// TwinCAT 3 PLC project LS21002
// ProgramVersion: 3.1.4023.0
// libraries:
//   Recipe Management, * (System)
//   SysMem, * (System)
//   Tc2_EtherCAT, * (Beckhoff Automation GmbH)
//   Tc2_Math, * (Beckhoff Automation GmbH)
//   Tc2_MC2, * (Beckhoff Automation GmbH)
//   Tc2_MC2_Drive, * (Beckhoff Automation GmbH)
//   Tc2_ModbusSrv, * (Beckhoff Automation GmbH)
//   Tc2_SPA, * (Beckhoff Automation GmbH)
//   Tc2_Standard, * (Beckhoff Automation GmbH)
//   Tc2_SUPS, * (Beckhoff Automation GmbH)
//   Tc2_System, * (Beckhoff Automation GmbH)
//   Tc2_TcpIp, * (Beckhoff Automation GmbH)
//   Tc2_Utilities, * (Beckhoff Automation GmbH)
//   Tc3_Module, * (Beckhoff Automation GmbH)
//   BASE,1.0.0.0,MEGA
// project tree:
//   DUTs/Camera/ DUT_CameraSend.TcDUT, DUT_CameraReceive.TcDUT, ST_CameraPara.TcDUT
//   DUTs/ DUT_NCIO.TcDUT, DUT_NCIO_1.TcDUT
//   DUTs/EPS Robot/ CmdRobot1.TcDUT, DUT_SysFromRobot1.TcDUT, DUT_SysToRobot1.TcDUT, stPutPartPosChoose.TcDUT, stTakePartPosChoose.TcDUT
//   DUTs/IO/ EL1889.TcDUT, EL2889.TcDUT
//   DUTs/Others/ DUT_Calibration.TcDUT, DUT_Sta.TcDUT, DUT_StaHistory.TcDUT, stEasyPumpsParamter.TcDUT, stWorkStatus.TcDUT, tDateAndTime.TcDUT
//   DUTs/PartData/ DUT_BeltLineFixture.TcDUT, DUT_LidChecking.TcDUT, DUT_MainlineFixture.TcDUT, DUT_PartFlag.TcDUT, DUT_PartStatus.TcDUT, DUT_PartStatus_1.TcDUT, DUT_Robot2.TcDUT, DUT_Process.TcDUT
//   DUTs/PartSequence/ tsPartSequence.TcDUT, tsSequence.TcDUT
//   DUTs/PC/ DUT_FomularData.TcDUT, DUT_PCReceive.TcDUT, DUT_PCSend.TcDUT, DUT_UploadProcessData.TcDUT
//   DUTs/Recipe/ DUT.TcDUT, ST_Thermostat.TcDUT
//   GVLs/ Common.TcGVL, GVL_Config.TcGVL, GVL_Robot.TcGVL, GVL_PC.TcGVL, GVL_Standard.TcGVL, GVL_System.TcGVL, GVL_UPS.TcGVL, IO.TcGVL
//   / PlcTask.TcTTO
//   POUs/001_Station/001_Mapping/ InputLink.TcPOU, OutputLink.TcPOU
//   POUs/001_Station/ S01_Loading.TcPOU, S02_LidInjecting.TcPOU, S03_LidChecking.TcPOU, S04_AluCovering.TcPOU, S05_Adjusting.TcPOU, S06_Cutting.TcPOU, S07_BoxCarrying.TcPOU, S08_MainLine.TcPOU, S09_CardCarrying.TcPOU, S10_BeltCarrying.TcPOU, S11_Packing.TcPOU, S12_PreLine.TcPOU, S13_Labeling.TcPOU, S14_LabelChecking.TcPOU, S15_NG.TcPOU, S16_Unloading.TcPOU
//   POUs/002_Machine/ CallStandard.TcPOU, CommWithPC.TcPOU, ControlMachine.TcPOU, LightsTest.TcPOU
//   POUs/003_FB/0000_FB_Alive/ FB_Alive.TcPOU
//   POUs/003_FB/0014_HITBOT/ HITBOT_ERROR.TcDUT, stCmdType.TcDUT, stHIBOTLocalPara.TcDUT, FB_ERG_20C.TcPOU, stDeviceStatus.TcDUT, stOper_Para.TcDUT, stReadPara.TcDUT, stRealPara.TcDUT, stSetPara.TcDUT
//   POUs/003_FB/0015_Functions/001_Parallel/ FC_ParallelFinished.TcPOU, FC_ParallelRequest.TcPOU
//   POUs/003_FB/0015_Functions/ FC_BubbleSort_Max.TcPOU, FC_BubbleSort_Min.TcPOU
//   POUs/003_FB/03_TURINRobotFB/DUTs/ CmdRobot.TcDUT, DUT_SysFromRobot.TcDUT, DUT_SysToRobot.TcDUT, ST_Sys_Para.TcDUT, ST_TURINROBOT_Data.TcDUT, TURIN_ERROR.TcDUT, TURIN_STATE.TcDUT, T_MaxString.TcDUT
//   POUs/003_FB/03_TURINRobotFB/ FB_TURINContorl.TcPOU
//   POUs/003_FB/0001_200Smart/ FB_Modbus_200Smart.TcPOU
//   POUs/003_FB/0001_200Smart/S7-200SMART/ DUT_200SMART.TcDUT (not stored)
//   POUs/003_FB/0002_Camera/ FB_Camera.TcPOU
//   POUs/003_FB/0003_EtherCATState/ FB_EtherCatSlaveMonitor.TcPOU (not stored)
//   POUs/003_FB/0004_FlowLine/ DUT_Motor.TcDUT (not stored), FB_FlowLine.TcPOU
//   POUs/003_FB/0005_EncoderCounter/ FB_Encoder.TcPOU (not stored)
//   POUs/003_FB/0006_ATV/ FB_ATV12.TcPOU
//   POUs/003_FB/0007_Vacuum/ FB_SmcVacuum.TcPOU
//   POUs/003_FB/05_StationFB/ E_State.TcDUT, FB_Station.TcPOU
//   POUs/003_FB/0008_LocalClient/ FB_LocalClient.TcPOU
//   POUs/003_FB/0009_MKC204C/DUTs/ MT_MCK_CMD.TcDUT, MT_MCK_ERROR.TcDUT, ST_DeviceOpe.TcDUT, ST_MCK_ParIn.TcDUT (not stored), ST_MCK_ParOut.TcDUT, ST_SysPar.TcDUT
//   POUs/003_FB/0009_MKC204C/ FB_MKC204C.TcPOU
//   POUs/003_FB/0010_LoadCell/ DUT_DeviceOpe.TcDUT, ST_LoadCell_Error.TcDUT (not stored), FB_LoadCell.TcPOU, FB_Modbus_Tcp.TcPOU, stModbusPara.TcDUT (not stored), ST_LoadCell_ParOut.TcDUT (not stored)
//   POUs/003_FB/0011_Cimcor/ FB_Cimcor_IZN10E.TcPOU
//   POUs/003_FB/0012_EasyPump/DUT/ PumpError.TcDUT, stEasyPumpHeadType.TcDUT, stEasyPumpHmi.TcDUT, stEasyPumpSoftType.TcDUT, stEasyPumpType.TcDUT, stOperType.TcDUT, st_EasyPump.TcDUT, ST_StepStatus.TcDUT, ST_LocalPara.TcDUT, ST_ReadPara.TcDUT, ST_SetPara.TcDUT
//   POUs/003_FB/0012_EasyPump/ FB_KF300.TcPOU
//   POUs/003_FB/0013_RGI_14_new/不带旋转的电动夹爪/ FB_RGI_14_Modbus.TcPOU
//   POUs/003_FB/0013_RGI_14_new/带旋转的电动夹爪/ FB_RGI_14_Modbus_1.TcPOU (not stored)
//   POUs/003_FB/100_test/12_BlinkFB/ FB_Blinker.TcPOU (not stored), ST_SysPulse.TcDUT (not stored)
//   POUs/003_FB/100_test/ FB_GetTime.TcPOU
//   POUs/003_FB/10_CylinderFB/ FB_Cylinder.TcPOU, ST_DataCylinder.TcDUT
//   POUs/003_FB/0013_RGI_14_new/ RGI_14_CMD.TcDUT (not stored), RGI_14_ERROR.TcDUT, ST_RGI_14_IOData.TcDUT (not stored), ST_RGI_14_Sys_Para.TcDUT, ST_RGI_HMIStates.TcDUT, ST_RGI_Opera.TcDUT, ST_RGI_PosPara.TcDUT
//   POUs/003_FB/14_MachineFB/ FB_Machine.TcPOU, ST_DataMachine.TcDUT, ST_OpeButton.TcDUT
//   POUs/003_FB/17_HMIFB/ FB_Proface.TcPOU
//   POUs/003_FB/19-AxisFB/ DUT_ActPos.TcDUT, FB_Axis.TcPOU, FB_AxisHome.TcPOU, FB_Axis_old.TcPOU, ST_DataAxis.TcDUT
//   POUs/003_FB/41_GetSystemTime/ DUT_TIMESET.TcDUT, PRG_GetSystemTime.TcPOU
//   POUs/003_FB/43_implicit checks/ CheckBounds.TcPOU, CheckDivDInt.TcPOU, CheckDivLInt.TcPOU, CheckDivLReal.TcPOU, CheckDivReal.TcPOU, CheckLRangeSigned.TcPOU, CheckLRangeUnsigned.TcPOU, CheckPointer.TcPOU, CheckRangeSigned.TcPOU, CheckRangeUnsigned.TcPOU
//   POUs/003_FB/0016_Recipe/ FB_Recipes.TcPOU (not stored), ST_Recipe.TcDUT
//   POUs/003_FB/064_Temperature/ FB_TempControl_FUSHI.TcPOU, ST_FUSHI_PXF_ParRead.TcDUT (not stored), ST_FUSHI_PXF_ParSet.TcDUT (not stored), ST_FUSHI_PXF_Sys_Pointer.TcDUT (not stored)
//   POUs/003_FB/53_RudongPump/08_PeristalticPumpFB/DUTs/ RudongPump_CMD.TcDUT, RudongPump_ERROR.TcDUT, RudongPump_IOData.TcDUT, RudongPump_Ope.TcDUT, RudongPump_PumpHeadType.TcDUT, RudongPump_PumpType.TcDUT, RudongPump_RunData.TcDUT, RudongPump_SoftPipeType.TcDUT, RudongPump_Sys_Para.TcDUT, STATE_1.TcDUT, ST_ModbusAddress.TcDUT
//   POUs/003_FB/53_RudongPump/08_PeristalticPumpFB/ FB_RuDongPump_modbus_DF600Plus.TcPOU, FB_RuDongPump_modbus_LABV.TcPOU
//   POUs/003_FB/53_RudongPump/08_PeristalticPumpFB/校准程序/ AutoCal_CMD.TcDUT, AutoCal_ERROR.TcDUT, FB_AutoCal.TcPOU, STAutoCal_ParIn.TcDUT, STAutoCal_ParOut.TcDUT, ST_AutoCalOpe.TcDUT, ST_AutoCal_SysPar.TcDUT
//   POUs/003_FB/53_RudongPump/08_PeristalticPumpFB/梅特勒托利多秤/ FB_MT_MKC.TcPOU
//   POUs/003_FB/53_RudongPump/09_PeristalticPumpFB/ FB_RuDongPump_ModbusTCP.TcPOU, RudongPump_CMD_1.TcDUT, RudongPump_ERROR_1.TcDUT, RudongPump_IOData_1.TcDUT, RuDongPump_ModbusAddress.TcDUT, RudongPump_Ope_1.TcDUT, RudongPump_PumpHeadType_1.TcDUT, RudongPump_PumpType_1.TcDUT, RudongPump_RunData_1.TcDUT, RudongPump_SoftPipeType_1.TcDUT, RudongPump_Sys_Para_1.TcDUT
//   POUs/003_FB/53_RudongPump/41 Modbus指令/DataExchange/ ModbusTCP_ErrorQuery.TcPOU
//   POUs/003_FB/53_RudongPump/41 Modbus指令/ FB_ModbusTCP.TcPOU, ModbusParIn.TcDUT, ModbusParOut.TcDUT, Modbus_Cmd.TcDUT, Modbus_ErrorCode.TcDUT, Modbus_Operation.TcDUT, Modbus_SysPar.TcDUT
//   POUs/003_FB/Z_ERG_20 FB/DUTs/ ERG_20_CMD.TcDUT, ERG_20_ERROR.TcDUT, ST_ERG_20_IOData.TcDUT, ST_ERG_20_Sys_Para.TcDUT, ST_Huiling_Pers_Para.TcDUT, ST_Huiling_PosPara.TcDUT
//   POUs/003_FB/Z_ERG_20 FB/ FB_ERG_20_Modbus.TcPOU
//   POUs/40_TcpIp/40_TcpIp/ E_ClientSteps.TcDUT, E_DataExchaSteps.TcDUT (not stored), FB_ClientDataExcha.TcPOU, FB_TcpIpClient.TcPOU (not stored), stTcpIpBaseParaCfg.TcDUT (not stored), TcpIpClientConstants.TcGVL
//   POUs/ MAIN.TcPOU, RecipeManager.TcRMO (not stored)
// real-time tasks:
//   TASK PlcTask: cycle T#10ms, priority 20, ADS port 350
// motion (NC):
//   TASK NC-Task 1 SAF: cycle T#2ms, priority 4, ADS port 501
//   TASK NC-Task 1 SVB: cycle T#10ms, priority 8, ADS port 511
//   AXIS Axis 1 (id 1)
//     PositionAreaControl: Enable=false
//     TargetPosControl: Enable=false
//     OtherSettings: AllowMotionCmdToSlave=true
//     encoder EncType=19
//       EncPara: ScaleFactorNumerator=20, ScaleFactorDenominator=4194304, MaxCount=#xffffffff
//     drive DrvType=16
//       DrvPara: MaxCount=#xffffffff, DriveControlDWord=#x00020100
//         Analog: TorqueSetpointScale=10, ScaleFactorActTorque=0.1
//         TimeComp: TaskDelayCycles=1
//     controller CtrType=1
//       CtrPara: PriorControlFactor=1
//         PosDiffControl: Enable=false
//         Observer: BandWidth=20
//   AXIS Axis 2 (id 2)
//     PositionAreaControl: Enable=false
//     TargetPosControl: Enable=false
//     OtherSettings: AllowMotionCmdToSlave=true
//     encoder EncType=19
//       EncPara: ScaleFactorNumerator=20, ScaleFactorDenominator=4194304, MaxCount=#xffffffff
//     drive DrvType=16
//       DrvPara: MaxCount=#xffffffff, DriveControlDWord=#x00020100
//         Analog: TorqueSetpointScale=10, ScaleFactorActTorque=0.1
//         TimeComp: TaskDelayCycles=1
//     controller CtrType=1
//       CtrPara: PriorControlFactor=1
//         PosDiffControl: Enable=false
//         Observer: BandWidth=20
//   AXIS Axis 3 (id 3)
//     PositionAreaControl: Enable=false
//     TargetPosControl: Enable=false
//     OtherSettings: AllowMotionCmdToSlave=true
//     encoder EncType=19
//       EncPara: ScaleFactorNumerator=20, ScaleFactorDenominator=4194304, MaxCount=#xffffffff
//     drive DrvType=16
//       DrvPara: MaxCount=#xffffffff, DriveControlDWord=#x00020100
//         Analog: TorqueSetpointScale=10, ScaleFactorActTorque=0.1
//         TimeComp: TaskDelayCycles=1
//     controller CtrType=1
//       CtrPara: PriorControlFactor=1
//         PosDiffControl: Enable=false
//         Observer: BandWidth=20
//   AXIS Axis 4 (id 4)
//     PositionAreaControl: Enable=false
//     TargetPosControl: Enable=false
//     OtherSettings: AllowMotionCmdToSlave=true
//     encoder EncType=19
//       EncPara: ScaleFactorNumerator=20, ScaleFactorDenominator=4194304, MaxCount=#xffffffff
//     drive DrvType=16
//       DrvPara: MaxCount=#xffffffff, DriveControlDWord=#x00020100
//         Analog: TorqueSetpointScale=10, ScaleFactorActTorque=0.1
//         TimeComp: TaskDelayCycles=1
//     controller CtrType=1
//       CtrPara: PriorControlFactor=1
//         PosDiffControl: Enable=false
//         Observer: BandWidth=20
//   AXIS Axis 5 (id 5)
//     PositionAreaControl: Enable=false
//     TargetPosControl: Enable=false
//     OtherSettings: AllowMotionCmdToSlave=true
//     encoder EncType=19
//       EncPara: ScaleFactorNumerator=5, ScaleFactorDenominator=4194304, MaxCount=#xffffffff
//     drive DrvType=16
//       DrvPara: MaxCount=#xffffffff, DriveControlDWord=#x00020100
//         Analog: TorqueSetpointScale=10, ScaleFactorActTorque=0.1
//         TimeComp: TaskDelayCycles=1
//     controller CtrType=1
//       CtrPara: PriorControlFactor=1
//         PosDiffControl: Enable=false
//         Observer: BandWidth=20
//   AXIS Axis 6 (id 6)
//     PositionAreaControl: Enable=false
//     TargetPosControl: Enable=false
//     OtherSettings: AllowMotionCmdToSlave=true
//     encoder EncType=19
//       EncPara: ScaleFactorNumerator=20, ScaleFactorDenominator=4194304, MaxCount=#xffffffff
//     drive DrvType=16
//       DrvPara: MaxCount=#xffffffff, DriveControlDWord=#x00020100
//         Analog: TorqueSetpointScale=10, ScaleFactorActTorque=0.1
//         TimeComp: TaskDelayCycles=1
//     controller CtrType=1
//       CtrPara: PriorControlFactor=1
//         PosDiffControl: Enable=false
//         Observer: BandWidth=20
//   AXIS Axis 7 (id 7)
//     PositionAreaControl: Enable=false
//     TargetPosControl: Enable=false
//     OtherSettings: AllowMotionCmdToSlave=true
//     encoder EncType=19
//       EncPara: ScaleFactorNumerator=20, ScaleFactorDenominator=4194304, MaxCount=#xffffffff
//     drive DrvType=16
//       DrvPara: MaxCount=#xffffffff, DriveControlDWord=#x00020100
//         Analog: TorqueSetpointScale=10, ScaleFactorActTorque=0.1
//         TimeComp: TaskDelayCycles=1
//     controller CtrType=1
//       CtrPara: PriorControlFactor=1
//         PosDiffControl: Enable=false
//         Observer: BandWidth=20
//   AXIS Axis 8 (id 8)
//     PositionAreaControl: Enable=false
//     TargetPosControl: Enable=false
//     OtherSettings: AllowMotionCmdToSlave=true
//     encoder EncType=19
//       EncPara: ScaleFactorNumerator=5, ScaleFactorDenominator=4194304, MaxCount=#xffffffff
//     drive DrvType=16
//       DrvPara: MaxCount=#xffffffff, DriveControlDWord=#x00020100
//         Analog: TorqueSetpointScale=10, ScaleFactorActTorque=0.1
//         TimeComp: TaskDelayCycles=1
//     controller CtrType=1
//       CtrPara: PriorControlFactor=1
//         PosDiffControl: Enable=false
//         Observer: BandWidth=20
//   AXIS Axis 9 (id 9)
//     PositionAreaControl: Enable=false
//     TargetPosControl: Enable=false
//     OtherSettings: AllowMotionCmdToSlave=true
//     encoder EncType=19
//       EncPara: ScaleFactorNumerator=18, ScaleFactorDenominator=4194304, MaxCount=#xffffffff
//     drive DrvType=16
//       DrvPara: MaxCount=#xffffffff, DriveControlDWord=#x00020100
//         Analog: TorqueSetpointScale=10, ScaleFactorActTorque=0.1
//         TimeComp: TaskDelayCycles=1
//     controller CtrType=1
//       CtrPara: PriorControlFactor=1
//         PosDiffControl: Enable=false
//         Observer: BandWidth=20
//   AXIS Axis 10 (id 10)
//     PositionAreaControl: Enable=false
//     TargetPosControl: Enable=false
//     OtherSettings: AllowMotionCmdToSlave=true
//     encoder EncType=19
//       EncPara: ScaleFactorNumerator=2, ScaleFactorDenominator=4194304, MaxCount=#xffffffff
//     drive DrvType=16
//       DrvPara: MaxCount=#xffffffff, DriveControlDWord=#x00020100
//         Analog: TorqueSetpointScale=10, ScaleFactorActTorque=0.1
//         TimeComp: TaskDelayCycles=1
//     controller CtrType=1
//       CtrPara: PriorControlFactor=1
//         PosDiffControl: Enable=false
//         Observer: BandWidth=20
//   AXIS Axis 11 (id 11)
//     PositionAreaControl: Enable=false
//     TargetPosControl: Enable=false
//     OtherSettings: AllowMotionCmdToSlave=true
//     encoder EncType=19
//       EncPara: ScaleFactorNumerator=2, ScaleFactorDenominator=4194304, MaxCount=#xffffffff
//     drive DrvType=16
//       DrvPara: MaxCount=#xffffffff, DriveControlDWord=#x00020100
//         Analog: TorqueSetpointScale=10, ScaleFactorActTorque=0.1
//         TimeComp: TaskDelayCycles=1
//     controller CtrType=1
//       CtrPara: PriorControlFactor=1
//         PosDiffControl: Enable=false
//         Observer: BandWidth=20
//   AXIS Axis 12 (id 12)
//     PositionAreaControl: Enable=false
//     TargetPosControl: Enable=false
//     OtherSettings: AllowMotionCmdToSlave=true
//     encoder EncType=19
//       EncPara: ScaleFactorNumerator=2, ScaleFactorDenominator=4194304, MaxCount=#xffffffff
//     drive DrvType=16
//       DrvPara: MaxCount=#xffffffff, DriveControlDWord=#x00020100
//         Analog: TorqueSetpointScale=10, ScaleFactorActTorque=0.1
//         TimeComp: TaskDelayCycles=1
//     controller CtrType=1
//       CtrPara: PriorControlFactor=1
//         PosDiffControl: Enable=false
//         Observer: BandWidth=20
//   AXIS Axis 13 (id 13)
//     PositionAreaControl: Enable=false
//     TargetPosControl: Enable=false
//     OtherSettings: AllowMotionCmdToSlave=true
//     encoder EncType=19
//       EncPara: ScaleFactorNumerator=2, ScaleFactorDenominator=4194304, MaxCount=#xffffffff
//     drive DrvType=16
//       DrvPara: MaxCount=#xffffffff, DriveControlDWord=#x00020100
//         Analog: TorqueSetpointScale=10, ScaleFactorActTorque=0.1
//         TimeComp: TaskDelayCycles=1
//     controller CtrType=1
//       CtrPara: PriorControlFactor=1
//         PosDiffControl: Enable=false
//         Observer: BandWidth=20
//   AXIS Axis 14 (id 14)
//     PositionAreaControl: Enable=false
//     TargetPosControl: Enable=false
//     OtherSettings: AllowMotionCmdToSlave=true
//     encoder EncType=19
//       EncPara: ScaleFactorNumerator=36, ScaleFactorDenominator=4194304, MaxCount=#xffffffff
//     drive DrvType=16
//       DrvPara: MaxCount=#xffffffff, DriveControlDWord=#x00020100
//         Analog: TorqueSetpointScale=10, ScaleFactorActTorque=0.1
//         TimeComp: TaskDelayCycles=1
//     controller CtrType=1
//       CtrPara: PriorControlFactor=1
//         PosDiffControl: Enable=false
//         Observer: BandWidth=20
//   AXIS Axis 15 (id 15)
//     PositionAreaControl: Enable=false
//     TargetPosControl: Enable=false
//     OtherSettings: AllowMotionCmdToSlave=true
//     encoder EncType=19
//       EncPara: ScaleFactorNumerator=18.22123708, ScaleFactorDenominator=4194304, MaxCount=#xffffffff
//     drive DrvType=16
//       DrvPara: MaxCount=#xffffffff, DriveControlDWord=#x00020100
//         Analog: TorqueSetpointScale=10, ScaleFactorActTorque=0.1
//         TimeComp: TaskDelayCycles=1
//     controller CtrType=1
//       CtrPara: PriorControlFactor=1
//         PosDiffControl: Enable=false
//         Observer: BandWidth=20
//   AXIS Axis 16 (id 16)
//     PositionAreaControl: Enable=false
//     TargetPosControl: Enable=false
//     OtherSettings: AllowMotionCmdToSlave=true
//     encoder EncType=19
//       EncPara: ScaleFactorNumerator=20, ScaleFactorDenominator=4194304, MaxCount=#xffffffff
//     drive DrvType=16
//       DrvPara: MaxCount=#xffffffff, DriveControlDWord=#x00020100
//         Analog: TorqueSetpointScale=10, ScaleFactorActTorque=0.1
//         TimeComp: TaskDelayCycles=1
//     controller CtrType=1
//       CtrPara: PriorControlFactor=1
//         PosDiffControl: Enable=false
//         Observer: BandWidth=20
//   AXIS Axis 17 (id 17)
//     PositionAreaControl: Enable=false
//     TargetPosControl: Enable=false
//     OtherSettings: AllowMotionCmdToSlave=true
//     encoder EncType=19
//       EncPara: ScaleFactorNumerator=10, ScaleFactorDenominator=12800, MaxCount=#xffffffff
//     drive DrvType=16
//       DrvPara: MaxCount=#xffffffff, DriveControlDWord=#x00020000
//         Analog: TorqueSetpointScale=10, ScaleFactorActTorque=0.1
//         TimeComp: TaskDelayCycles=1
//     controller CtrType=1
//       CtrPara: PriorControlFactor=1
//         PosDiffControl: Enable=false
//         Observer: BandWidth=20
//   AXIS Axis 18 (id 18)
//     PositionAreaControl: Enable=false
//     TargetPosControl: Enable=false
//     OtherSettings: AllowMotionCmdToSlave=true
//     encoder EncType=19
//       EncPara: ScaleFactorNumerator=10, ScaleFactorDenominator=12800, MaxCount=#xffffffff
//     drive DrvType=16
//       DrvPara: MaxCount=#xffffffff, DriveControlDWord=#x00020000
//         Analog: TorqueSetpointScale=10, ScaleFactorActTorque=0.1
//         TimeComp: TaskDelayCycles=1
//     controller CtrType=1
//       CtrPara: PriorControlFactor=1
//         PosDiffControl: Enable=false
//         Observer: BandWidth=20
//   AXIS Axis 19 (id 19)
//     PositionAreaControl: Enable=false
//     TargetPosControl: Enable=false
//     OtherSettings: AllowMotionCmdToSlave=true
//     encoder EncType=19
//       EncPara: ScaleFactorNumerator=10, ScaleFactorDenominator=12800, MaxCount=#xffffffff
//     drive DrvType=16
//       DrvPara: MaxCount=#xffffffff, DriveControlDWord=#x00020000
//         Analog: TorqueSetpointScale=10, ScaleFactorActTorque=0.1
//         TimeComp: TaskDelayCycles=1
//     controller CtrType=1
//       CtrPara: PriorControlFactor=1
//         PosDiffControl: Enable=false
//         Observer: BandWidth=20
// I/O:
//   DEVICE Device 1 (EtherCAT), AmsNetId 192.168.1.1.2.1
//     Term 16 (EK1200) [EK1200-5000 EtherCAT Power supply (2A E-Bus)]
//       Term 2 (EL1889) [EL1889 16Ch. Dig. Input 24V, 3ms, negative]
//       Term 3 (EL1889) [EL1889 16Ch. Dig. Input 24V, 3ms, negative]
//       Term 4 (EL1889) [EL1889 16Ch. Dig. Input 24V, 3ms, negative]
//       Term 5 (EL1889) [EL1889 16Ch. Dig. Input 24V, 3ms, negative]
//       Term 6 (EL1889) [EL1889 16Ch. Dig. Input 24V, 3ms, negative]
//       Term 7 (EL1889) [EL1889 16Ch. Dig. Input 24V, 3ms, negative]
//       Term 8 (EL2889) [EL2889 16Ch. Dig. Output 24V, 0.5A, negative]
//       Term 9 (EL2889) [EL2889 16Ch. Dig. Output 24V, 0.5A, negative]
//       Term 25 (EL2889) [EL2889 16Ch. Dig. Output 24V, 0.5A, negative]
//       Term 26 (EL2889) [EL2889 16Ch. Dig. Output 24V, 0.5A, negative]
//       Term 27 (EL2889) [EL2889 16Ch. Dig. Output 24V, 0.5A, negative]
//       Term 28 (EL2889) [EL2889 16Ch. Dig. Output 24V, 0.5A, negative]
//       Term 29 (EK1122) [EK1122 2 port EtherCAT junction]
//         Drive 30 (MR-JET-G-N1) [MR-JET-G-N1 EtherCAT Drive (CoE) ver.B9]
//         Drive 31 (MR-JET-G-N1) [MR-JET-G-N1 EtherCAT Drive (CoE) ver.B9]
//         Drive 32 (MR-JET-G-N1) [MR-JET-G-N1 EtherCAT Drive (CoE) ver.B9]
//         Drive 33 (MR-JET-G-N1) [MR-JET-G-N1 EtherCAT Drive (CoE) ver.B9]
//         Drive 34 (MR-JET-G-N1) [MR-JET-G-N1 EtherCAT Drive (CoE) ver.C0]
//         Drive 35 (MR-JET-G-N1) [MR-JET-G-N1 EtherCAT Drive (CoE) ver.B9]
//         Drive 36 (MR-JET-G-N1) [MR-JET-G-N1 EtherCAT Drive (CoE) ver.B9]
//         Drive 37 (MR-JET-G-N1) [MR-JET-G-N1 EtherCAT Drive (CoE) ver.C0]
//         Term 38 (EK1100) [EK1100 EtherCAT Coupler (2A E-Bus)]
//           Term 39 (EL1889) [EL1889 16Ch. Dig. Input 24V, 3ms, negative]
//           Term 73 (EL2889) [EL2889 16Ch. Dig. Output 24V, 0.5A, negative]
//           Term 62 (EL9011) [EL9011 End Terminal]
//         Drive 40 (MR-JET-G-N1) [MR-JET-G-N1 EtherCAT Drive (CoE) ver.B9]
//         Term 41 (EK1100) [EK1100 EtherCAT Coupler (2A E-Bus)]
//           Term 42 (EL1889) [EL1889 16Ch. Dig. Input 24V, 3ms, negative]
//           Term 43 (EL1889) [EL1889 16Ch. Dig. Input 24V, 3ms, negative]
//           Term 44 (EL1889) [EL1889 16Ch. Dig. Input 24V, 3ms, negative]
//           Term 45 (EL1889) [EL1889 16Ch. Dig. Input 24V, 3ms, negative]
//           Term 46 (EL1889) [EL1889 16Ch. Dig. Input 24V, 3ms, negative]
//           Term 47 (EL1889) [EL1889 16Ch. Dig. Input 24V, 3ms, negative]
//           Term 48 (EL2889) [EL2889 16Ch. Dig. Output 24V, 0.5A, negative]
//           Term 49 (EL2889) [EL2889 16Ch. Dig. Output 24V, 0.5A, negative]
//           Term 50 (EL2889) [EL2889 16Ch. Dig. Output 24V, 0.5A, negative]
//           Term 51 (EL2889) [EL2889 16Ch. Dig. Output 24V, 0.5A, negative]
//           Term 63 (EL9011) [EL9011 End Terminal]
//         Drive 52 (MR-JET-G-N1) [MR-JET-G-N1 EtherCAT Drive (CoE) ver.C0]
//         Drive 53 (MR-JET-G-N1) [MR-JET-G-N1 EtherCAT Drive (CoE) ver.C0]
//         Drive 54 (MR-JET-G-N1) [MR-JET-G-N1 EtherCAT Drive (CoE) ver.C0]
//         Drive 55 (MR-JET-G-N1) [MR-JET-G-N1 EtherCAT Drive (CoE) ver.C0]
//         Drive 56 (MR-JET-G-N1) [MR-JET-G-N1 EtherCAT Drive (CoE) ver.C0]
//         Drive 57 (MR-JET-G-N1) [MR-JET-G-N1 EtherCAT Drive (CoE) ver.C0]
//         Drive 58 (MR-JET-G-N1) [MR-JET-G-N1 EtherCAT Drive (CoE) ver.B9]
//         Drive 59 (DM3C-EC556) [DM3C-EC556(COE)]
//         Drive 60 (DM3C-EC556) [DM3C-EC556(COE)]
//         Drive 61 (DM3C-EC870) [DM3C-EC870(COE)]
//         Term 95 (EK1100) [EK1100 EtherCAT Coupler (2A E-Bus)]
//           Term 96 (EL1889) [EL1889 16Ch. Dig. Input 24V, 3ms, negative]
//           Term 97 (EL1889) [EL1889 16Ch. Dig. Input 24V, 3ms, negative]
//           Term 98 (EL2889) [EL2889 16Ch. Dig. Output 24V, 0.5A, negative]
//           Term 99 (EL2889) [EL2889 16Ch. Dig. Output 24V, 0.5A, negative]
//           Term 103 (EL9011) [EL9011 End Terminal]
//         Box 100 (GR10-2HCE) [GR10-2HCE_1.4.5.0]
//   DEVICE Device 2 (EtherCAT Automation Protocol), AmsNetId 192.168.1.1.3.1
//   DEVICE Device 3 (EtherCAT Automation Protocol), AmsNetId 192.168.1.1.4.1
//   DEVICE Device 4 (COM Port)
// variable links:
//   NC-Task 1 SAF/Axes/Axis 1 <-> Device 1 (EtherCAT)/Term 16 (EK1200)/Term 29 (EK1122)/Drive 30 (MR-JET-G-N1)
//     Drive/Inputs/In/nDataIn1 <-> 1st Transmit PDO Mapping/Following error actual value
//     Drive/Inputs/In/nDataIn3[0] <-> 1st Transmit PDO Mapping/Torque actual value
//     Drive/Inputs/In/nDcOutputTime <-> InfoData/DcOutputShift
//     Drive/Inputs/In/nState1 <-> 1st Transmit PDO Mapping/Statusword
//     Drive/Inputs/In/nState2 <-> 1st Transmit PDO Mapping/Statusword @bit 8
//     Drive/Inputs/In/nState4 @bit 1 <-> WcState/InputToggle
//     Drive/Inputs/In/nState4 <-> WcState/WcState
//     Drive/Inputs/In/nState5 <-> 1st Transmit PDO Mapping/Modes of operation display
//     Drive/Outputs/Out/nDataOut1 <-> 1st Receive PDO Mapping/Target position
//     Drive/Outputs/Out/nDataOut2 <-> 1st Receive PDO Mapping/Target velocity
//     Drive/Outputs/Out/nDataOut4[0] <-> 1st Receive PDO Mapping/Target torque
//     Enc/Inputs/In/nDataIn1 <-> 1st Transmit PDO Mapping/Position actual value
//     Enc/Inputs/In/nDataIn7 <-> 1st Transmit PDO Mapping/Velocity actual value
//     Enc/Inputs/In/nDcInputTime <-> InfoData/DcInputShift
//     Enc/Inputs/In/nState4 @bit 1 <-> WcState/InputToggle
//     Enc/Inputs/In/nState4 <-> WcState/WcState
//   NC-Task 1 SAF/Axes/Axis 10 <-> Device 1 (EtherCAT)/Term 16 (EK1200)/Term 29 (EK1122)/Drive 52 (MR-JET-G-N1)
//     Drive/Inputs/In/nDataIn1 <-> 1st Transmit PDO Mapping/Following error actual value
//     Drive/Inputs/In/nDataIn3[0] <-> 1st Transmit PDO Mapping/Torque actual value
//     Drive/Inputs/In/nDcOutputTime <-> InfoData/DcOutputShift
//     Drive/Inputs/In/nState1 <-> 1st Transmit PDO Mapping/Statusword
//     Drive/Inputs/In/nState2 <-> 1st Transmit PDO Mapping/Statusword @bit 8
//     Drive/Inputs/In/nState4 @bit 1 <-> WcState/InputToggle
//     Drive/Inputs/In/nState4 <-> WcState/WcState
//     Drive/Inputs/In/nState5 <-> 1st Transmit PDO Mapping/Modes of operation display
//     Drive/Outputs/Out/nDataOut1 <-> 1st Receive PDO Mapping/Target position
//     Drive/Outputs/Out/nDataOut2 <-> 1st Receive PDO Mapping/Target velocity
//     Drive/Outputs/Out/nDataOut4[0] <-> 1st Receive PDO Mapping/Target torque
//     Enc/Inputs/In/nDataIn1 <-> 1st Transmit PDO Mapping/Position actual value
//     Enc/Inputs/In/nDataIn7 <-> 1st Transmit PDO Mapping/Velocity actual value
//     Enc/Inputs/In/nDcInputTime <-> InfoData/DcInputShift
//     Enc/Inputs/In/nState4 @bit 1 <-> WcState/InputToggle
//     Enc/Inputs/In/nState4 <-> WcState/WcState
//   NC-Task 1 SAF/Axes/Axis 11 <-> Device 1 (EtherCAT)/Term 16 (EK1200)/Term 29 (EK1122)/Drive 53 (MR-JET-G-N1)
//     Drive/Inputs/In/nDataIn1 <-> 1st Transmit PDO Mapping/Following error actual value
//     Drive/Inputs/In/nDataIn3[0] <-> 1st Transmit PDO Mapping/Torque actual value
//     Drive/Inputs/In/nDcOutputTime <-> InfoData/DcOutputShift
//     Drive/Inputs/In/nState1 <-> 1st Transmit PDO Mapping/Statusword
//     Drive/Inputs/In/nState2 <-> 1st Transmit PDO Mapping/Statusword @bit 8
//     Drive/Inputs/In/nState4 @bit 1 <-> WcState/InputToggle
//     Drive/Inputs/In/nState4 <-> WcState/WcState
//     Drive/Inputs/In/nState5 <-> 1st Transmit PDO Mapping/Modes of operation display
//     Drive/Outputs/Out/nDataOut1 <-> 1st Receive PDO Mapping/Target position
//     Drive/Outputs/Out/nDataOut2 <-> 1st Receive PDO Mapping/Target velocity
//     Drive/Outputs/Out/nDataOut4[0] <-> 1st Receive PDO Mapping/Target torque
//     Enc/Inputs/In/nDataIn1 <-> 1st Transmit PDO Mapping/Position actual value
//     Enc/Inputs/In/nDataIn7 <-> 1st Transmit PDO Mapping/Velocity actual value
//     Enc/Inputs/In/nDcInputTime <-> InfoData/DcInputShift
//     Enc/Inputs/In/nState4 @bit 1 <-> WcState/InputToggle
//     Enc/Inputs/In/nState4 <-> WcState/WcState
//   NC-Task 1 SAF/Axes/Axis 12 <-> Device 1 (EtherCAT)/Term 16 (EK1200)/Term 29 (EK1122)/Drive 54 (MR-JET-G-N1)
//     Drive/Inputs/In/nDataIn1 <-> 1st Transmit PDO Mapping/Following error actual value
//     Drive/Inputs/In/nDataIn3[0] <-> 1st Transmit PDO Mapping/Torque actual value
//     Drive/Inputs/In/nDcOutputTime <-> InfoData/DcOutputShift
//     Drive/Inputs/In/nState1 <-> 1st Transmit PDO Mapping/Statusword
//     Drive/Inputs/In/nState2 <-> 1st Transmit PDO Mapping/Statusword @bit 8
//     Drive/Inputs/In/nState4 @bit 1 <-> WcState/InputToggle
//     Drive/Inputs/In/nState4 <-> WcState/WcState
//     Drive/Inputs/In/nState5 <-> 1st Transmit PDO Mapping/Modes of operation display
//     Drive/Outputs/Out/nDataOut1 <-> 1st Receive PDO Mapping/Target position
//     Drive/Outputs/Out/nDataOut2 <-> 1st Receive PDO Mapping/Target velocity
//     Drive/Outputs/Out/nDataOut4[0] <-> 1st Receive PDO Mapping/Target torque
//     Enc/Inputs/In/nDataIn1 <-> 1st Transmit PDO Mapping/Position actual value
//     Enc/Inputs/In/nDataIn7 <-> 1st Transmit PDO Mapping/Velocity actual value
//     Enc/Inputs/In/nDcInputTime <-> InfoData/DcInputShift
//     Enc/Inputs/In/nState4 @bit 1 <-> WcState/InputToggle
//     Enc/Inputs/In/nState4 <-> WcState/WcState
//   NC-Task 1 SAF/Axes/Axis 13 <-> Device 1 (EtherCAT)/Term 16 (EK1200)/Term 29 (EK1122)/Drive 55 (MR-JET-G-N1)
//     Drive/Inputs/In/nDataIn1 <-> 1st Transmit PDO Mapping/Following error actual value
//     Drive/Inputs/In/nDataIn3[0] <-> 1st Transmit PDO Mapping/Torque actual value
//     Drive/Inputs/In/nDcOutputTime <-> InfoData/DcOutputShift
//     Drive/Inputs/In/nState1 <-> 1st Transmit PDO Mapping/Statusword
//     Drive/Inputs/In/nState2 <-> 1st Transmit PDO Mapping/Statusword @bit 8
//     Drive/Inputs/In/nState4 @bit 1 <-> WcState/InputToggle
//     Drive/Inputs/In/nState4 <-> WcState/WcState
//     Drive/Inputs/In/nState5 <-> 1st Transmit PDO Mapping/Modes of operation display
//     Drive/Outputs/Out/nDataOut1 <-> 1st Receive PDO Mapping/Target position
//     Drive/Outputs/Out/nDataOut2 <-> 1st Receive PDO Mapping/Target velocity
//     Drive/Outputs/Out/nDataOut4[0] <-> 1st Receive PDO Mapping/Target torque
//     Enc/Inputs/In/nDataIn1 <-> 1st Transmit PDO Mapping/Position actual value
//     Enc/Inputs/In/nDataIn7 <-> 1st Transmit PDO Mapping/Velocity actual value
//     Enc/Inputs/In/nDcInputTime <-> InfoData/DcInputShift
//     Enc/Inputs/In/nState4 @bit 1 <-> WcState/InputToggle
//     Enc/Inputs/In/nState4 <-> WcState/WcState
//   NC-Task 1 SAF/Axes/Axis 14 <-> Device 1 (EtherCAT)/Term 16 (EK1200)/Term 29 (EK1122)/Drive 56 (MR-JET-G-N1)
//     Drive/Inputs/In/nDataIn1 <-> 1st Transmit PDO Mapping/Following error actual value
//     Drive/Inputs/In/nDataIn3[0] <-> 1st Transmit PDO Mapping/Torque actual value
//     Drive/Inputs/In/nDcOutputTime <-> InfoData/DcOutputShift
//     Drive/Inputs/In/nState1 <-> 1st Transmit PDO Mapping/Statusword
//     Drive/Inputs/In/nState2 <-> 1st Transmit PDO Mapping/Statusword @bit 8
//     Drive/Inputs/In/nState4 @bit 1 <-> WcState/InputToggle
//     Drive/Inputs/In/nState4 <-> WcState/WcState
//     Drive/Inputs/In/nState5 <-> 1st Transmit PDO Mapping/Modes of operation display
//     Drive/Outputs/Out/nDataOut1 <-> 1st Receive PDO Mapping/Target position
//     Drive/Outputs/Out/nDataOut2 <-> 1st Receive PDO Mapping/Target velocity
//     Drive/Outputs/Out/nDataOut4[0] <-> 1st Receive PDO Mapping/Target torque
//     Enc/Inputs/In/nDataIn1 <-> 1st Transmit PDO Mapping/Position actual value
//     Enc/Inputs/In/nDataIn7 <-> 1st Transmit PDO Mapping/Velocity actual value
//     Enc/Inputs/In/nDcInputTime <-> InfoData/DcInputShift
//     Enc/Inputs/In/nState4 @bit 1 <-> WcState/InputToggle
//     Enc/Inputs/In/nState4 <-> WcState/WcState
//   NC-Task 1 SAF/Axes/Axis 15 <-> Device 1 (EtherCAT)/Term 16 (EK1200)/Term 29 (EK1122)/Drive 57 (MR-JET-G-N1)
//     Drive/Inputs/In/nDataIn1 <-> 1st Transmit PDO Mapping/Following error actual value
//     Drive/Inputs/In/nDataIn3[0] <-> 1st Transmit PDO Mapping/Torque actual value
//     Drive/Inputs/In/nDcOutputTime <-> InfoData/DcOutputShift
//     Drive/Inputs/In/nState1 <-> 1st Transmit PDO Mapping/Statusword
//     Drive/Inputs/In/nState2 <-> 1st Transmit PDO Mapping/Statusword @bit 8
//     Drive/Inputs/In/nState4 @bit 1 <-> WcState/InputToggle
//     Drive/Inputs/In/nState4 <-> WcState/WcState
//     Drive/Inputs/In/nState5 <-> 1st Transmit PDO Mapping/Modes of operation display
//     Drive/Outputs/Out/nDataOut1 <-> 1st Receive PDO Mapping/Target position
//     Drive/Outputs/Out/nDataOut2 <-> 1st Receive PDO Mapping/Target velocity
//     Drive/Outputs/Out/nDataOut4[0] <-> 1st Receive PDO Mapping/Target torque
//     Enc/Inputs/In/nDataIn1 <-> 1st Transmit PDO Mapping/Position actual value
//     Enc/Inputs/In/nDataIn7 <-> 1st Transmit PDO Mapping/Velocity actual value
//     Enc/Inputs/In/nDcInputTime <-> InfoData/DcInputShift
//     Enc/Inputs/In/nState4 @bit 1 <-> WcState/InputToggle
//     Enc/Inputs/In/nState4 <-> WcState/WcState
//   NC-Task 1 SAF/Axes/Axis 16 <-> Device 1 (EtherCAT)/Term 16 (EK1200)/Term 29 (EK1122)/Drive 58 (MR-JET-G-N1)
//     Drive/Inputs/In/nDataIn1 <-> 1st Transmit PDO Mapping/Following error actual value
//     Drive/Inputs/In/nDataIn3[0] <-> 1st Transmit PDO Mapping/Torque actual value
//     Drive/Inputs/In/nDcOutputTime <-> InfoData/DcOutputShift
//     Drive/Inputs/In/nState1 <-> 1st Transmit PDO Mapping/Statusword
//     Drive/Inputs/In/nState2 <-> 1st Transmit PDO Mapping/Statusword @bit 8
//     Drive/Inputs/In/nState4 @bit 1 <-> WcState/InputToggle
//     Drive/Inputs/In/nState4 <-> WcState/WcState
//     Drive/Inputs/In/nState5 <-> 1st Transmit PDO Mapping/Modes of operation display
//     Drive/Outputs/Out/nDataOut1 <-> 1st Receive PDO Mapping/Target position
//     Drive/Outputs/Out/nDataOut2 <-> 1st Receive PDO Mapping/Target velocity
//     Drive/Outputs/Out/nDataOut4[0] <-> 1st Receive PDO Mapping/Target torque
//     Enc/Inputs/In/nDataIn1 <-> 1st Transmit PDO Mapping/Position actual value
//     Enc/Inputs/In/nDataIn7 <-> 1st Transmit PDO Mapping/Velocity actual value
//     Enc/Inputs/In/nDcInputTime <-> InfoData/DcInputShift
//     Enc/Inputs/In/nState4 @bit 1 <-> WcState/InputToggle
//     Enc/Inputs/In/nState4 <-> WcState/WcState
//   NC-Task 1 SAF/Axes/Axis 17 <-> Device 1 (EtherCAT)/Term 16 (EK1200)/Term 29 (EK1122)/Drive 59 (DM3C-EC556)
//     Drive/Inputs/In/nDcOutputTime <-> InfoData/DcOutputShift
//     Drive/Inputs/In/nState1 <-> Transmit PDO 1/Status Word
//     Drive/Inputs/In/nState2 <-> Transmit PDO 1/Status Word @bit 8
//     Drive/Inputs/In/nState4 @bit 1 <-> WcState/InputToggle
//     Drive/Inputs/In/nState4 <-> WcState/WcState
//     Drive/Inputs/In/nState5 <-> Transmit PDO 1/Modes of Operation display
//     Drive/Outputs/Out/nDataOut1 <-> Receive PDO 1/Profile Target Position
//     Enc/Inputs/In/nDataIn1 <-> Transmit PDO 1/Position Actual Value
//     Enc/Inputs/In/nDataIn3 <-> Transmit PDO 1/Touch Probe 1 Positive Value
//     Enc/Inputs/In/nDcInputTime <-> InfoData/DcInputShift
//     Enc/Inputs/In/nState4 @bit 1 <-> WcState/InputToggle
//     Enc/Inputs/In/nState4 <-> WcState/WcState
//     Enc/Inputs/In/nState5 <-> Transmit PDO 1/Touch Probe Status
//     Enc/Inputs/In/nState6 <-> Transmit PDO 1/Touch Probe Status @bit 8
//     Enc/Outputs/Out/nCtrl5 <-> Receive PDO 1/Touch Probe Function
//     Enc/Outputs/Out/nCtrl6 <-> Receive PDO 1/Touch Probe Function @bit 8
//   NC-Task 1 SAF/Axes/Axis 18 <-> Device 1 (EtherCAT)/Term 16 (EK1200)/Term 29 (EK1122)/Drive 60 (DM3C-EC556)
//     Drive/Inputs/In/nDcOutputTime <-> InfoData/DcOutputShift
//     Drive/Inputs/In/nState1 <-> Transmit PDO 1/Status Word
//     Drive/Inputs/In/nState2 <-> Transmit PDO 1/Status Word @bit 8
//     Drive/Inputs/In/nState4 @bit 1 <-> WcState/InputToggle
//     Drive/Inputs/In/nState4 <-> WcState/WcState
//     Drive/Inputs/In/nState5 <-> Transmit PDO 1/Modes of Operation display
//     Drive/Outputs/Out/nDataOut1 <-> Receive PDO 1/Profile Target Position
//     Enc/Inputs/In/nDataIn1 <-> Transmit PDO 1/Position Actual Value
//     Enc/Inputs/In/nDataIn3 <-> Transmit PDO 1/Touch Probe 1 Positive Value
//     Enc/Inputs/In/nDcInputTime <-> InfoData/DcInputShift
//     Enc/Inputs/In/nState4 @bit 1 <-> WcState/InputToggle
//     Enc/Inputs/In/nState4 <-> WcState/WcState
//     Enc/Inputs/In/nState5 <-> Transmit PDO 1/Touch Probe Status
//     Enc/Inputs/In/nState6 <-> Transmit PDO 1/Touch Probe Status @bit 8
//     Enc/Outputs/Out/nCtrl5 <-> Receive PDO 1/Touch Probe Function
//     Enc/Outputs/Out/nCtrl6 <-> Receive PDO 1/Touch Probe Function @bit 8
//   NC-Task 1 SAF/Axes/Axis 19 <-> Device 1 (EtherCAT)/Term 16 (EK1200)/Term 29 (EK1122)/Drive 61 (DM3C-EC870)
//     Drive/Inputs/In/nDcOutputTime <-> InfoData/DcOutputShift
//     Drive/Inputs/In/nState1 <-> Transmit PDO 1/Status Word
//     Drive/Inputs/In/nState2 <-> Transmit PDO 1/Status Word @bit 8
//     Drive/Inputs/In/nState4 @bit 1 <-> WcState/InputToggle
//     Drive/Inputs/In/nState4 <-> WcState/WcState
//     Drive/Inputs/In/nState5 <-> Transmit PDO 1/Modes of Operation display
//     Drive/Outputs/Out/nDataOut1 <-> Receive PDO 1/Profile Target Position
//     Enc/Inputs/In/nDataIn1 <-> Transmit PDO 1/Position Actual Value
//     Enc/Inputs/In/nDataIn3 <-> Transmit PDO 1/Touch Probe 1 Positive Value
//     Enc/Inputs/In/nDcInputTime <-> InfoData/DcInputShift
//     Enc/Inputs/In/nState4 @bit 1 <-> WcState/InputToggle
//     Enc/Inputs/In/nState4 <-> WcState/WcState
//     Enc/Inputs/In/nState5 <-> Transmit PDO 1/Touch Probe Status
//     Enc/Inputs/In/nState6 <-> Transmit PDO 1/Touch Probe Status @bit 8
//     Enc/Outputs/Out/nCtrl5 <-> Receive PDO 1/Touch Probe Function
//     Enc/Outputs/Out/nCtrl6 <-> Receive PDO 1/Touch Probe Function @bit 8
//   NC-Task 1 SAF/Axes/Axis 2 <-> Device 1 (EtherCAT)/Term 16 (EK1200)/Term 29 (EK1122)/Drive 31 (MR-JET-G-N1)
//     Drive/Inputs/In/nDataIn1 <-> 1st Transmit PDO Mapping/Following error actual value
//     Drive/Inputs/In/nDataIn3[0] <-> 1st Transmit PDO Mapping/Torque actual value
//     Drive/Inputs/In/nDcOutputTime <-> InfoData/DcOutputShift
//     Drive/Inputs/In/nState1 <-> 1st Transmit PDO Mapping/Statusword
//     Drive/Inputs/In/nState2 <-> 1st Transmit PDO Mapping/Statusword @bit 8
//     Drive/Inputs/In/nState4 @bit 1 <-> WcState/InputToggle
//     Drive/Inputs/In/nState4 <-> WcState/WcState
//     Drive/Inputs/In/nState5 <-> 1st Transmit PDO Mapping/Modes of operation display
//     Drive/Outputs/Out/nDataOut1 <-> 1st Receive PDO Mapping/Target position
//     Drive/Outputs/Out/nDataOut2 <-> 1st Receive PDO Mapping/Target velocity
//     Drive/Outputs/Out/nDataOut4[0] <-> 1st Receive PDO Mapping/Target torque
//     Enc/Inputs/In/nDataIn1 <-> 1st Transmit PDO Mapping/Position actual value
//     Enc/Inputs/In/nDataIn7 <-> 1st Transmit PDO Mapping/Velocity actual value
//     Enc/Inputs/In/nDcInputTime <-> InfoData/DcInputShift
//     Enc/Inputs/In/nState4 @bit 1 <-> WcState/InputToggle
//     Enc/Inputs/In/nState4 <-> WcState/WcState
//   NC-Task 1 SAF/Axes/Axis 3 <-> Device 1 (EtherCAT)/Term 16 (EK1200)/Term 29 (EK1122)/Drive 32 (MR-JET-G-N1)
//     Drive/Inputs/In/nDataIn1 <-> 1st Transmit PDO Mapping/Following error actual value
//     Drive/Inputs/In/nDataIn3[0] <-> 1st Transmit PDO Mapping/Torque actual value
//     Drive/Inputs/In/nDcOutputTime <-> InfoData/DcOutputShift
//     Drive/Inputs/In/nState1 <-> 1st Transmit PDO Mapping/Statusword
//     Drive/Inputs/In/nState2 <-> 1st Transmit PDO Mapping/Statusword @bit 8
//     Drive/Inputs/In/nState4 @bit 1 <-> WcState/InputToggle
//     Drive/Inputs/In/nState4 <-> WcState/WcState
//     Drive/Inputs/In/nState5 <-> 1st Transmit PDO Mapping/Modes of operation display
//     Drive/Outputs/Out/nDataOut1 <-> 1st Receive PDO Mapping/Target position
//     Drive/Outputs/Out/nDataOut2 <-> 1st Receive PDO Mapping/Target velocity
//     Drive/Outputs/Out/nDataOut4[0] <-> 1st Receive PDO Mapping/Target torque
//     Enc/Inputs/In/nDataIn1 <-> 1st Transmit PDO Mapping/Position actual value
//     Enc/Inputs/In/nDataIn7 <-> 1st Transmit PDO Mapping/Velocity actual value
//     Enc/Inputs/In/nDcInputTime <-> InfoData/DcInputShift
//     Enc/Inputs/In/nState4 @bit 1 <-> WcState/InputToggle
//     Enc/Inputs/In/nState4 <-> WcState/WcState
//   NC-Task 1 SAF/Axes/Axis 4 <-> Device 1 (EtherCAT)/Term 16 (EK1200)/Term 29 (EK1122)/Drive 33 (MR-JET-G-N1)
//     Drive/Inputs/In/nDataIn1 <-> 1st Transmit PDO Mapping/Following error actual value
//     Drive/Inputs/In/nDataIn3[0] <-> 1st Transmit PDO Mapping/Torque actual value
//     Drive/Inputs/In/nDcOutputTime <-> InfoData/DcOutputShift
//     Drive/Inputs/In/nState1 <-> 1st Transmit PDO Mapping/Statusword
//     Drive/Inputs/In/nState2 <-> 1st Transmit PDO Mapping/Statusword @bit 8
//     Drive/Inputs/In/nState4 @bit 1 <-> WcState/InputToggle
//     Drive/Inputs/In/nState4 <-> WcState/WcState
//     Drive/Inputs/In/nState5 <-> 1st Transmit PDO Mapping/Modes of operation display
//     Drive/Outputs/Out/nDataOut1 <-> 1st Receive PDO Mapping/Target position
//     Drive/Outputs/Out/nDataOut2 <-> 1st Receive PDO Mapping/Target velocity
//     Drive/Outputs/Out/nDataOut4[0] <-> 1st Receive PDO Mapping/Target torque
//     Enc/Inputs/In/nDataIn1 <-> 1st Transmit PDO Mapping/Position actual value
//     Enc/Inputs/In/nDataIn7 <-> 1st Transmit PDO Mapping/Velocity actual value
//     Enc/Inputs/In/nDcInputTime <-> InfoData/DcInputShift
//     Enc/Inputs/In/nState4 @bit 1 <-> WcState/InputToggle
//     Enc/Inputs/In/nState4 <-> WcState/WcState
//   NC-Task 1 SAF/Axes/Axis 5 <-> Device 1 (EtherCAT)/Term 16 (EK1200)/Term 29 (EK1122)/Drive 34 (MR-JET-G-N1)
//     Drive/Inputs/In/nDataIn1 <-> 1st Transmit PDO Mapping/Following error actual value
//     Drive/Inputs/In/nDataIn3[0] <-> 1st Transmit PDO Mapping/Torque actual value
//     Drive/Inputs/In/nDcOutputTime <-> InfoData/DcOutputShift
//     Drive/Inputs/In/nState1 <-> 1st Transmit PDO Mapping/Statusword
//     Drive/Inputs/In/nState2 <-> 1st Transmit PDO Mapping/Statusword @bit 8
//     Drive/Inputs/In/nState4 @bit 1 <-> WcState/InputToggle
//     Drive/Inputs/In/nState4 <-> WcState/WcState
//     Drive/Inputs/In/nState5 <-> 1st Transmit PDO Mapping/Modes of operation display
//     Drive/Outputs/Out/nDataOut1 <-> 1st Receive PDO Mapping/Target position
//     Drive/Outputs/Out/nDataOut2 <-> 1st Receive PDO Mapping/Target velocity
//     Drive/Outputs/Out/nDataOut4[0] <-> 1st Receive PDO Mapping/Target torque
//     Enc/Inputs/In/nDataIn1 <-> 1st Transmit PDO Mapping/Position actual value
//     Enc/Inputs/In/nDataIn7 <-> 1st Transmit PDO Mapping/Velocity actual value
//     Enc/Inputs/In/nDcInputTime <-> InfoData/DcInputShift
//     Enc/Inputs/In/nState4 @bit 1 <-> WcState/InputToggle
//     Enc/Inputs/In/nState4 <-> WcState/WcState
//   NC-Task 1 SAF/Axes/Axis 6 <-> Device 1 (EtherCAT)/Term 16 (EK1200)/Term 29 (EK1122)/Drive 35 (MR-JET-G-N1)
//     Drive/Inputs/In/nDataIn1 <-> 1st Transmit PDO Mapping/Following error actual value
//     Drive/Inputs/In/nDataIn3[0] <-> 1st Transmit PDO Mapping/Torque actual value
//     Drive/Inputs/In/nDcOutputTime <-> InfoData/DcOutputShift
//     Drive/Inputs/In/nState1 <-> 1st Transmit PDO Mapping/Statusword
//     Drive/Inputs/In/nState2 <-> 1st Transmit PDO Mapping/Statusword @bit 8
//     Drive/Inputs/In/nState4 @bit 1 <-> WcState/InputToggle
//     Drive/Inputs/In/nState4 <-> WcState/WcState
//     Drive/Inputs/In/nState5 <-> 1st Transmit PDO Mapping/Modes of operation display
//     Drive/Outputs/Out/nDataOut1 <-> 1st Receive PDO Mapping/Target position
//     Drive/Outputs/Out/nDataOut2 <-> 1st Receive PDO Mapping/Target velocity
//     Drive/Outputs/Out/nDataOut4[0] <-> 1st Receive PDO Mapping/Target torque
//     Enc/Inputs/In/nDataIn1 <-> 1st Transmit PDO Mapping/Position actual value
//     Enc/Inputs/In/nDataIn7 <-> 1st Transmit PDO Mapping/Velocity actual value
//     Enc/Inputs/In/nDcInputTime <-> InfoData/DcInputShift
//     Enc/Inputs/In/nState4 @bit 1 <-> WcState/InputToggle
//     Enc/Inputs/In/nState4 <-> WcState/WcState
//   NC-Task 1 SAF/Axes/Axis 7 <-> Device 1 (EtherCAT)/Term 16 (EK1200)/Term 29 (EK1122)/Drive 36 (MR-JET-G-N1)
//     Drive/Inputs/In/nDataIn1 <-> 1st Transmit PDO Mapping/Following error actual value
//     Drive/Inputs/In/nDataIn3[0] <-> 1st Transmit PDO Mapping/Torque actual value
//     Drive/Inputs/In/nDcOutputTime <-> InfoData/DcOutputShift
//     Drive/Inputs/In/nState1 <-> 1st Transmit PDO Mapping/Statusword
//     Drive/Inputs/In/nState2 <-> 1st Transmit PDO Mapping/Statusword @bit 8
//     Drive/Inputs/In/nState4 @bit 1 <-> WcState/InputToggle
//     Drive/Inputs/In/nState4 <-> WcState/WcState
//     Drive/Inputs/In/nState5 <-> 1st Transmit PDO Mapping/Modes of operation display
//     Drive/Outputs/Out/nDataOut1 <-> 1st Receive PDO Mapping/Target position
//     Drive/Outputs/Out/nDataOut2 <-> 1st Receive PDO Mapping/Target velocity
//     Drive/Outputs/Out/nDataOut4[0] <-> 1st Receive PDO Mapping/Target torque
//     Enc/Inputs/In/nDataIn1 <-> 1st Transmit PDO Mapping/Position actual value
//     Enc/Inputs/In/nDataIn7 <-> 1st Transmit PDO Mapping/Velocity actual value
//     Enc/Inputs/In/nDcInputTime <-> InfoData/DcInputShift
//     Enc/Inputs/In/nState4 @bit 1 <-> WcState/InputToggle
//     Enc/Inputs/In/nState4 <-> WcState/WcState
//   NC-Task 1 SAF/Axes/Axis 8 <-> Device 1 (EtherCAT)/Term 16 (EK1200)/Term 29 (EK1122)/Drive 37 (MR-JET-G-N1)
//     Drive/Inputs/In/nDataIn1 <-> 1st Transmit PDO Mapping/Following error actual value
//     Drive/Inputs/In/nDataIn3[0] <-> 1st Transmit PDO Mapping/Torque actual value
//     Drive/Inputs/In/nDcOutputTime <-> InfoData/DcOutputShift
//     Drive/Inputs/In/nState1 <-> 1st Transmit PDO Mapping/Statusword
//     Drive/Inputs/In/nState2 <-> 1st Transmit PDO Mapping/Statusword @bit 8
//     Drive/Inputs/In/nState4 @bit 1 <-> WcState/InputToggle
//     Drive/Inputs/In/nState4 <-> WcState/WcState
//     Drive/Inputs/In/nState5 <-> 1st Transmit PDO Mapping/Modes of operation display
//     Drive/Outputs/Out/nDataOut1 <-> 1st Receive PDO Mapping/Target position
//     Drive/Outputs/Out/nDataOut2 <-> 1st Receive PDO Mapping/Target velocity
//     Drive/Outputs/Out/nDataOut4[0] <-> 1st Receive PDO Mapping/Target torque
//     Enc/Inputs/In/nDataIn1 <-> 1st Transmit PDO Mapping/Position actual value
//     Enc/Inputs/In/nDataIn7 <-> 1st Transmit PDO Mapping/Velocity actual value
//     Enc/Inputs/In/nDcInputTime <-> InfoData/DcInputShift
//     Enc/Inputs/In/nState4 @bit 1 <-> WcState/InputToggle
//     Enc/Inputs/In/nState4 <-> WcState/WcState
//   NC-Task 1 SAF/Axes/Axis 9 <-> Device 1 (EtherCAT)/Term 16 (EK1200)/Term 29 (EK1122)/Drive 40 (MR-JET-G-N1)
//     Drive/Inputs/In/nDataIn1 <-> 1st Transmit PDO Mapping/Following error actual value
//     Drive/Inputs/In/nDataIn3[0] <-> 1st Transmit PDO Mapping/Torque actual value
//     Drive/Inputs/In/nDcOutputTime <-> InfoData/DcOutputShift
//     Drive/Inputs/In/nState1 <-> 1st Transmit PDO Mapping/Statusword
//     Drive/Inputs/In/nState2 <-> 1st Transmit PDO Mapping/Statusword @bit 8
//     Drive/Inputs/In/nState4 @bit 1 <-> WcState/InputToggle
//     Drive/Inputs/In/nState4 <-> WcState/WcState
//     Drive/Inputs/In/nState5 <-> 1st Transmit PDO Mapping/Modes of operation display
//     Drive/Outputs/Out/nDataOut1 <-> 1st Receive PDO Mapping/Target position
//     Drive/Outputs/Out/nDataOut2 <-> 1st Receive PDO Mapping/Target velocity
//     Drive/Outputs/Out/nDataOut4[0] <-> 1st Receive PDO Mapping/Target torque
//     Enc/Inputs/In/nDataIn1 <-> 1st Transmit PDO Mapping/Position actual value
//     Enc/Inputs/In/nDataIn7 <-> 1st Transmit PDO Mapping/Velocity actual value
//     Enc/Inputs/In/nDcInputTime <-> InfoData/DcInputShift
//     Enc/Inputs/In/nState4 @bit 1 <-> WcState/InputToggle
//     Enc/Inputs/In/nState4 <-> WcState/WcState
//   LS21002/LS21002 Instance <-> Device 1 (EtherCAT)/Term 16 (EK1200)/Term 2 (EL1889)
//     PlcTask Inputs/GVL_Standard.fbEhterCATSlaveMonitor[1].axIState[1] <-> WcState/WcState
//     PlcTask Inputs/IO.ET01_Input[1] @bit 9 <-> Channel 10/Input
//     PlcTask Inputs/IO.ET01_Input[1] @bit 10 <-> Channel 11/Input
//     PlcTask Inputs/IO.ET01_Input[1] @bit 11 <-> Channel 12/Input
//     PlcTask Inputs/IO.ET01_Input[1] @bit 12 <-> Channel 13/Input
//     PlcTask Inputs/IO.ET01_Input[1] @bit 13 <-> Channel 14/Input
//     PlcTask Inputs/IO.ET01_Input[1] @bit 14 <-> Channel 15/Input
//     PlcTask Inputs/IO.ET01_Input[1] @bit 15 <-> Channel 16/Input
//     PlcTask Inputs/IO.ET01_Input[1] @bit 1 <-> Channel 2/Input
//     PlcTask Inputs/IO.ET01_Input[1] @bit 2 <-> Channel 3/Input
//     PlcTask Inputs/IO.ET01_Input[1] @bit 3 <-> Channel 4/Input
//     PlcTask Inputs/IO.ET01_Input[1] @bit 4 <-> Channel 5/Input
//     PlcTask Inputs/IO.ET01_Input[1] @bit 5 <-> Channel 6/Input
//     PlcTask Inputs/IO.ET01_Input[1] @bit 6 <-> Channel 7/Input
//     PlcTask Inputs/IO.ET01_Input[1] @bit 7 <-> Channel 8/Input
//     PlcTask Inputs/IO.ET01_Input[1] @bit 8 <-> Channel 9/Input
//     PlcTask Inputs/IO.ET01_Input[1] <-> Channel 1/Input
//   LS21002/LS21002 Instance <-> Device 1 (EtherCAT)/Term 16 (EK1200)/Term 25 (EL2889)
//     PlcTask Inputs/GVL_Standard.fbEhterCATSlaveMonitor[1].axIState[9] <-> WcState/WcState
//     PlcTask Outputs/IO.ET01_Output[3] @bit 9 <-> Channel 10/Output
//     PlcTask Outputs/IO.ET01_Output[3] @bit 10 <-> Channel 11/Output
//     PlcTask Outputs/IO.ET01_Output[3] @bit 11 <-> Channel 12/Output
//     PlcTask Outputs/IO.ET01_Output[3] @bit 12 <-> Channel 13/Output
//     PlcTask Outputs/IO.ET01_Output[3] @bit 13 <-> Channel 14/Output
//     PlcTask Outputs/IO.ET01_Output[3] @bit 14 <-> Channel 15/Output
//     PlcTask Outputs/IO.ET01_Output[3] @bit 15 <-> Channel 16/Output
//     PlcTask Outputs/IO.ET01_Output[3] @bit 1 <-> Channel 2/Output
//     PlcTask Outputs/IO.ET01_Output[3] @bit 2 <-> Channel 3/Output
//     PlcTask Outputs/IO.ET01_Output[3] @bit 3 <-> Channel 4/Output
//     PlcTask Outputs/IO.ET01_Output[3] @bit 4 <-> Channel 5/Output
//     PlcTask Outputs/IO.ET01_Output[3] @bit 5 <-> Channel 6/Output
//     PlcTask Outputs/IO.ET01_Output[3] @bit 6 <-> Channel 7/Output
//     PlcTask Outputs/IO.ET01_Output[3] @bit 7 <-> Channel 8/Output
//     PlcTask Outputs/IO.ET01_Output[3] @bit 8 <-> Channel 9/Output
//     PlcTask Outputs/IO.ET01_Output[3] <-> Channel 1/Output
//   LS21002/LS21002 Instance <-> Device 1 (EtherCAT)/Term 16 (EK1200)/Term 26 (EL2889)
//     PlcTask Inputs/GVL_Standard.fbEhterCATSlaveMonitor[1].axIState[10] <-> WcState/WcState
//     PlcTask Outputs/IO.ET01_Output[4] @bit 9 <-> Channel 10/Output
//     PlcTask Outputs/IO.ET01_Output[4] @bit 10 <-> Channel 11/Output
//     PlcTask Outputs/IO.ET01_Output[4] @bit 11 <-> Channel 12/Output
//     PlcTask Outputs/IO.ET01_Output[4] @bit 12 <-> Channel 13/Output
//     PlcTask Outputs/IO.ET01_Output[4] @bit 13 <-> Channel 14/Output
//     PlcTask Outputs/IO.ET01_Output[4] @bit 14 <-> Channel 15/Output
//     PlcTask Outputs/IO.ET01_Output[4] @bit 15 <-> Channel 16/Output
//     PlcTask Outputs/IO.ET01_Output[4] @bit 1 <-> Channel 2/Output
//     PlcTask Outputs/IO.ET01_Output[4] @bit 2 <-> Channel 3/Output
//     PlcTask Outputs/IO.ET01_Output[4] @bit 3 <-> Channel 4/Output
//     PlcTask Outputs/IO.ET01_Output[4] @bit 4 <-> Channel 5/Output
//     PlcTask Outputs/IO.ET01_Output[4] @bit 5 <-> Channel 6/Output
//     PlcTask Outputs/IO.ET01_Output[4] @bit 6 <-> Channel 7/Output
//     PlcTask Outputs/IO.ET01_Output[4] @bit 7 <-> Channel 8/Output
//     PlcTask Outputs/IO.ET01_Output[4] @bit 8 <-> Channel 9/Output
//     PlcTask Outputs/IO.ET01_Output[4] <-> Channel 1/Output
//   LS21002/LS21002 Instance <-> Device 1 (EtherCAT)/Term 16 (EK1200)/Term 27 (EL2889)
//     PlcTask Inputs/GVL_Standard.fbEhterCATSlaveMonitor[1].axIState[11] <-> WcState/WcState
//     PlcTask Outputs/IO.ET01_Output[5] @bit 9 <-> Channel 10/Output
//     PlcTask Outputs/IO.ET01_Output[5] @bit 10 <-> Channel 11/Output
//     PlcTask Outputs/IO.ET01_Output[5] @bit 11 <-> Channel 12/Output
//     PlcTask Outputs/IO.ET01_Output[5] @bit 12 <-> Channel 13/Output
//     PlcTask Outputs/IO.ET01_Output[5] @bit 13 <-> Channel 14/Output
//     PlcTask Outputs/IO.ET01_Output[5] @bit 14 <-> Channel 15/Output
//     PlcTask Outputs/IO.ET01_Output[5] @bit 15 <-> Channel 16/Output
//     PlcTask Outputs/IO.ET01_Output[5] @bit 1 <-> Channel 2/Output
//     PlcTask Outputs/IO.ET01_Output[5] @bit 2 <-> Channel 3/Output
//     PlcTask Outputs/IO.ET01_Output[5] @bit 3 <-> Channel 4/Output
//     PlcTask Outputs/IO.ET01_Output[5] @bit 4 <-> Channel 5/Output
//     PlcTask Outputs/IO.ET01_Output[5] @bit 5 <-> Channel 6/Output
//     PlcTask Outputs/IO.ET01_Output[5] @bit 6 <-> Channel 7/Output
//     PlcTask Outputs/IO.ET01_Output[5] @bit 7 <-> Channel 8/Output
//     PlcTask Outputs/IO.ET01_Output[5] @bit 8 <-> Channel 9/Output
//     PlcTask Outputs/IO.ET01_Output[5] <-> Channel 1/Output
//   LS21002/LS21002 Instance <-> Device 1 (EtherCAT)/Term 16 (EK1200)/Term 28 (EL2889)
//     PlcTask Inputs/GVL_Standard.fbEhterCATSlaveMonitor[1].axIState[12] <-> WcState/WcState
//     PlcTask Outputs/IO.ET01_Output[6] @bit 9 <-> Channel 10/Output
//     PlcTask Outputs/IO.ET01_Output[6] @bit 10 <-> Channel 11/Output
//     PlcTask Outputs/IO.ET01_Output[6] @bit 11 <-> Channel 12/Output
//     PlcTask Outputs/IO.ET01_Output[6] @bit 12 <-> Channel 13/Output
//     PlcTask Outputs/IO.ET01_Output[6] @bit 13 <-> Channel 14/Output
//     PlcTask Outputs/IO.ET01_Output[6] @bit 14 <-> Channel 15/Output
//     PlcTask Outputs/IO.ET01_Output[6] @bit 15 <-> Channel 16/Output
//     PlcTask Outputs/IO.ET01_Output[6] @bit 1 <-> Channel 2/Output
//     PlcTask Outputs/IO.ET01_Output[6] @bit 2 <-> Channel 3/Output
//     PlcTask Outputs/IO.ET01_Output[6] @bit 3 <-> Channel 4/Output
//     PlcTask Outputs/IO.ET01_Output[6] @bit 4 <-> Channel 5/Output
//     PlcTask Outputs/IO.ET01_Output[6] @bit 5 <-> Channel 6/Output
//     PlcTask Outputs/IO.ET01_Output[6] @bit 6 <-> Channel 7/Output
//     PlcTask Outputs/IO.ET01_Output[6] @bit 7 <-> Channel 8/Output
//     PlcTask Outputs/IO.ET01_Output[6] @bit 8 <-> Channel 9/Output
//     PlcTask Outputs/IO.ET01_Output[6] <-> Channel 1/Output
//   LS21002/LS21002 Instance <-> Device 1 (EtherCAT)/Term 16 (EK1200)/Term 29 (EK1122)/Box 100 (GR10-2HCE)
//     PlcTask Inputs/GVL_Standard.fbEhterCATSlaveMonitor[4].axIState[5] <-> WcState/WcState
//     PlcTask Inputs/GVL_Standard.fbEncoder.IudiCounterValue <-> Ch1 TPDO Mapping Parameter/Ch1 encoder present position
//     PlcTask Outputs/GVL_Standard.fbEncoder.QiCounterCmd <-> Ch1 RPDO Mapping parameter 0/Ch1 encoder counter operation command
//   LS21002/LS21002 Instance <-> Device 1 (EtherCAT)/Term 16 (EK1200)/Term 29 (EK1122)/Drive 30 (MR-JET-G-N1)
//     PlcTask Inputs/GVL_Standard.arAxisSensor[1] <-> 1st Transmit PDO Mapping/Digital inputs
//     PlcTask Outputs/CallStandard.controlword[1] <-> 1st Receive PDO Mapping/Controlword
//     PlcTask Outputs/CallStandard.sModeOperation[1] <-> 1st Receive PDO Mapping/Modes of operation
//   LS21002/LS21002 Instance <-> Device 1 (EtherCAT)/Term 16 (EK1200)/Term 29 (EK1122)/Drive 31 (MR-JET-G-N1)
//     PlcTask Inputs/GVL_Standard.arAxisSensor[2] <-> 1st Transmit PDO Mapping/Digital inputs
//     PlcTask Outputs/CallStandard.controlword[2] <-> 1st Receive PDO Mapping/Controlword
//     PlcTask Outputs/CallStandard.sModeOperation[2] <-> 1st Receive PDO Mapping/Modes of operation
//   LS21002/LS21002 Instance <-> Device 1 (EtherCAT)/Term 16 (EK1200)/Term 29 (EK1122)/Drive 32 (MR-JET-G-N1)
//     PlcTask Inputs/GVL_Standard.arAxisSensor[3] <-> 1st Transmit PDO Mapping/Digital inputs
//     PlcTask Outputs/CallStandard.controlword[3] <-> 1st Receive PDO Mapping/Controlword
//     PlcTask Outputs/CallStandard.sModeOperation[3] <-> 1st Receive PDO Mapping/Modes of operation
//   LS21002/LS21002 Instance <-> Device 1 (EtherCAT)/Term 16 (EK1200)/Term 29 (EK1122)/Drive 33 (MR-JET-G-N1)
//     PlcTask Inputs/GVL_Standard.arAxisSensor[4] <-> 1st Transmit PDO Mapping/Digital inputs
//     PlcTask Outputs/CallStandard.controlword[4] <-> 1st Receive PDO Mapping/Controlword
//     PlcTask Outputs/CallStandard.sModeOperation[4] <-> 1st Receive PDO Mapping/Modes of operation
//   LS21002/LS21002 Instance <-> Device 1 (EtherCAT)/Term 16 (EK1200)/Term 29 (EK1122)/Drive 34 (MR-JET-G-N1)
//     PlcTask Inputs/GVL_Standard.arAxisSensor[5] <-> 1st Transmit PDO Mapping/Digital inputs
//     PlcTask Outputs/CallStandard.controlword[5] <-> 1st Receive PDO Mapping/Controlword
//     PlcTask Outputs/CallStandard.sModeOperation[5] <-> 1st Receive PDO Mapping/Modes of operation
//   LS21002/LS21002 Instance <-> Device 1 (EtherCAT)/Term 16 (EK1200)/Term 29 (EK1122)/Drive 35 (MR-JET-G-N1)
//     PlcTask Inputs/GVL_Standard.arAxisSensor[6] <-> 1st Transmit PDO Mapping/Digital inputs
//     PlcTask Outputs/CallStandard.controlword[6] <-> 1st Receive PDO Mapping/Controlword
//     PlcTask Outputs/CallStandard.sModeOperation[6] <-> 1st Receive PDO Mapping/Modes of operation
//   LS21002/LS21002 Instance <-> Device 1 (EtherCAT)/Term 16 (EK1200)/Term 29 (EK1122)/Drive 36 (MR-JET-G-N1)
//     PlcTask Inputs/GVL_Standard.arAxisSensor[7] <-> 1st Transmit PDO Mapping/Digital inputs
//     PlcTask Outputs/CallStandard.controlword[7] <-> 1st Receive PDO Mapping/Controlword
//     PlcTask Outputs/CallStandard.sModeOperation[7] <-> 1st Receive PDO Mapping/Modes of operation
//   LS21002/LS21002 Instance <-> Device 1 (EtherCAT)/Term 16 (EK1200)/Term 29 (EK1122)/Drive 37 (MR-JET-G-N1)
//     PlcTask Inputs/GVL_Standard.arAxisSensor[8] <-> 1st Transmit PDO Mapping/Digital inputs
//     PlcTask Outputs/CallStandard.controlword[8] <-> 1st Receive PDO Mapping/Controlword
//     PlcTask Outputs/CallStandard.sModeOperation[8] <-> 1st Receive PDO Mapping/Modes of operation
//   LS21002/LS21002 Instance <-> Device 1 (EtherCAT)/Term 16 (EK1200)/Term 29 (EK1122)/Drive 40 (MR-JET-G-N1)
//     PlcTask Inputs/GVL_Standard.arAxisSensor[9] <-> 1st Transmit PDO Mapping/Digital inputs
//     PlcTask Outputs/CallStandard.controlword[9] <-> 1st Receive PDO Mapping/Controlword
//     PlcTask Outputs/CallStandard.sModeOperation[9] <-> 1st Receive PDO Mapping/Modes of operation
//   LS21002/LS21002 Instance <-> Device 1 (EtherCAT)/Term 16 (EK1200)/Term 29 (EK1122)/Drive 52 (MR-JET-G-N1)
//     PlcTask Inputs/GVL_Standard.arAxisSensor[10] <-> 1st Transmit PDO Mapping/Digital inputs
//     PlcTask Outputs/CallStandard.controlword[10] <-> 1st Receive PDO Mapping/Controlword
//     PlcTask Outputs/CallStandard.sModeOperation[10] <-> 1st Receive PDO Mapping/Modes of operation
//   LS21002/LS21002 Instance <-> Device 1 (EtherCAT)/Term 16 (EK1200)/Term 29 (EK1122)/Drive 53 (MR-JET-G-N1)
//     PlcTask Inputs/GVL_Standard.arAxisSensor[11] <-> 1st Transmit PDO Mapping/Digital inputs
//     PlcTask Outputs/CallStandard.controlword[11] <-> 1st Receive PDO Mapping/Controlword
//     PlcTask Outputs/CallStandard.sModeOperation[11] <-> 1st Receive PDO Mapping/Modes of operation
//   LS21002/LS21002 Instance <-> Device 1 (EtherCAT)/Term 16 (EK1200)/Term 29 (EK1122)/Drive 54 (MR-JET-G-N1)
//     PlcTask Inputs/GVL_Standard.arAxisSensor[12] <-> 1st Transmit PDO Mapping/Digital inputs
//     PlcTask Outputs/CallStandard.controlword[12] <-> 1st Receive PDO Mapping/Controlword
//     PlcTask Outputs/CallStandard.sModeOperation[12] <-> 1st Receive PDO Mapping/Modes of operation
//   LS21002/LS21002 Instance <-> Device 1 (EtherCAT)/Term 16 (EK1200)/Term 29 (EK1122)/Drive 55 (MR-JET-G-N1)
//     PlcTask Inputs/GVL_Standard.arAxisSensor[13] <-> 1st Transmit PDO Mapping/Digital inputs
//     PlcTask Outputs/CallStandard.controlword[13] <-> 1st Receive PDO Mapping/Controlword
//     PlcTask Outputs/CallStandard.sModeOperation[13] <-> 1st Receive PDO Mapping/Modes of operation
//   LS21002/LS21002 Instance <-> Device 1 (EtherCAT)/Term 16 (EK1200)/Term 29 (EK1122)/Drive 56 (MR-JET-G-N1)
//     PlcTask Inputs/GVL_Standard.arAxisSensor[14] <-> 1st Transmit PDO Mapping/Digital inputs
//     PlcTask Outputs/CallStandard.controlword[14] <-> 1st Receive PDO Mapping/Controlword
//     PlcTask Outputs/CallStandard.sModeOperation[14] <-> 1st Receive PDO Mapping/Modes of operation
//   LS21002/LS21002 Instance <-> Device 1 (EtherCAT)/Term 16 (EK1200)/Term 29 (EK1122)/Drive 57 (MR-JET-G-N1)
//     PlcTask Inputs/GVL_Standard.arAxisSensor[15] <-> 1st Transmit PDO Mapping/Digital inputs
//     PlcTask Outputs/CallStandard.controlword[15] <-> 1st Receive PDO Mapping/Controlword
//     PlcTask Outputs/CallStandard.sModeOperation[15] <-> 1st Receive PDO Mapping/Modes of operation
//   LS21002/LS21002 Instance <-> Device 1 (EtherCAT)/Term 16 (EK1200)/Term 29 (EK1122)/Drive 58 (MR-JET-G-N1)
//     PlcTask Inputs/GVL_Standard.arAxisSensor[16] <-> 1st Transmit PDO Mapping/Digital inputs
//     PlcTask Outputs/CallStandard.controlword[16] <-> 1st Receive PDO Mapping/Controlword
//     PlcTask Outputs/CallStandard.sModeOperation[16] <-> 1st Receive PDO Mapping/Modes of operation
//   LS21002/LS21002 Instance <-> Device 1 (EtherCAT)/Term 16 (EK1200)/Term 29 (EK1122)/Drive 59 (DM3C-EC556)
//     PlcTask Inputs/GVL_Standard.arAxisSensor[17] <-> Transmit PDO 1/Digital Inputs
//     PlcTask Outputs/CallStandard.controlword[17] <-> Receive PDO 1/Control Word
//     PlcTask Outputs/CallStandard.sModeOperation[17] <-> Receive PDO 1/Modes of Operation
//   LS21002/LS21002 Instance <-> Device 1 (EtherCAT)/Term 16 (EK1200)/Term 29 (EK1122)/Drive 60 (DM3C-EC556)
//     PlcTask Inputs/GVL_Standard.arAxisSensor[18] <-> Transmit PDO 1/Digital Inputs
//     PlcTask Outputs/CallStandard.controlword[18] <-> Receive PDO 1/Control Word
//     PlcTask Outputs/CallStandard.sModeOperation[18] <-> Receive PDO 1/Modes of Operation
//   LS21002/LS21002 Instance <-> Device 1 (EtherCAT)/Term 16 (EK1200)/Term 29 (EK1122)/Drive 61 (DM3C-EC870)
//     PlcTask Inputs/GVL_Standard.arAxisSensor[19] <-> Transmit PDO 1/Digital Inputs
//     PlcTask Outputs/CallStandard.controlword[19] <-> Receive PDO 1/Control Word
//     PlcTask Outputs/CallStandard.sModeOperation[19] <-> Receive PDO 1/Modes of Operation
//   LS21002/LS21002 Instance <-> Device 1 (EtherCAT)/Term 16 (EK1200)/Term 29 (EK1122)/Term 38 (EK1100)/Term 39 (EL1889)
//     PlcTask Inputs/GVL_Standard.fbEhterCATSlaveMonitor[3].axIState[1] <-> WcState/WcState
//     PlcTask Inputs/IO.ET03_Input @bit 9 <-> Channel 10/Input
//     PlcTask Inputs/IO.ET03_Input @bit 10 <-> Channel 11/Input
//     PlcTask Inputs/IO.ET03_Input @bit 11 <-> Channel 12/Input
//     PlcTask Inputs/IO.ET03_Input @bit 12 <-> Channel 13/Input
//     PlcTask Inputs/IO.ET03_Input @bit 13 <-> Channel 14/Input
//     PlcTask Inputs/IO.ET03_Input @bit 14 <-> Channel 15/Input
//     PlcTask Inputs/IO.ET03_Input @bit 15 <-> Channel 16/Input
//     PlcTask Inputs/IO.ET03_Input @bit 1 <-> Channel 2/Input
//     PlcTask Inputs/IO.ET03_Input @bit 2 <-> Channel 3/Input
//     PlcTask Inputs/IO.ET03_Input @bit 3 <-> Channel 4/Input
//     PlcTask Inputs/IO.ET03_Input @bit 4 <-> Channel 5/Input
//     PlcTask Inputs/IO.ET03_Input @bit 5 <-> Channel 6/Input
//     PlcTask Inputs/IO.ET03_Input @bit 6 <-> Channel 7/Input
//     PlcTask Inputs/IO.ET03_Input @bit 7 <-> Channel 8/Input
//     PlcTask Inputs/IO.ET03_Input @bit 8 <-> Channel 9/Input
//     PlcTask Inputs/IO.ET03_Input <-> Channel 1/Input
//   LS21002/LS21002 Instance <-> Device 1 (EtherCAT)/Term 16 (EK1200)/Term 29 (EK1122)/Term 38 (EK1100)/Term 73 (EL2889)
//     PlcTask Outputs/IO.ET03_Output[1] @bit 9 <-> Channel 10/Output
//     PlcTask Outputs/IO.ET03_Output[1] @bit 10 <-> Channel 11/Output
//     PlcTask Outputs/IO.ET03_Output[1] @bit 11 <-> Channel 12/Output
//     PlcTask Outputs/IO.ET03_Output[1] @bit 12 <-> Channel 13/Output
//     PlcTask Outputs/IO.ET03_Output[1] @bit 13 <-> Channel 14/Output
//     PlcTask Outputs/IO.ET03_Output[1] @bit 14 <-> Channel 15/Output
//     PlcTask Outputs/IO.ET03_Output[1] @bit 15 <-> Channel 16/Output
//     PlcTask Outputs/IO.ET03_Output[1] @bit 1 <-> Channel 2/Output
//     PlcTask Outputs/IO.ET03_Output[1] @bit 2 <-> Channel 3/Output
//     PlcTask Outputs/IO.ET03_Output[1] @bit 3 <-> Channel 4/Output
//     PlcTask Outputs/IO.ET03_Output[1] @bit 4 <-> Channel 5/Output
//     PlcTask Outputs/IO.ET03_Output[1] @bit 5 <-> Channel 6/Output
//     PlcTask Outputs/IO.ET03_Output[1] @bit 6 <-> Channel 7/Output
//     PlcTask Outputs/IO.ET03_Output[1] @bit 7 <-> Channel 8/Output
//     PlcTask Outputs/IO.ET03_Output[1] @bit 8 <-> Channel 9/Output
//     PlcTask Outputs/IO.ET03_Output[1] <-> Channel 1/Output
//   LS21002/LS21002 Instance <-> Device 1 (EtherCAT)/Term 16 (EK1200)/Term 29 (EK1122)/Term 41 (EK1100)/Term 42 (EL1889)
//     PlcTask Inputs/GVL_Standard.fbEhterCATSlaveMonitor[2].axIState[1] <-> WcState/WcState
//     PlcTask Inputs/IO.ET02_Input[1] @bit 9 <-> Channel 10/Input
//     PlcTask Inputs/IO.ET02_Input[1] @bit 10 <-> Channel 11/Input
//     PlcTask Inputs/IO.ET02_Input[1] @bit 11 <-> Channel 12/Input
//     PlcTask Inputs/IO.ET02_Input[1] @bit 12 <-> Channel 13/Input
//     PlcTask Inputs/IO.ET02_Input[1] @bit 13 <-> Channel 14/Input
//     PlcTask Inputs/IO.ET02_Input[1] @bit 14 <-> Channel 15/Input
//     PlcTask Inputs/IO.ET02_Input[1] @bit 15 <-> Channel 16/Input
//     PlcTask Inputs/IO.ET02_Input[1] @bit 1 <-> Channel 2/Input
//     PlcTask Inputs/IO.ET02_Input[1] @bit 2 <-> Channel 3/Input
//     PlcTask Inputs/IO.ET02_Input[1] @bit 3 <-> Channel 4/Input
//     PlcTask Inputs/IO.ET02_Input[1] @bit 4 <-> Channel 5/Input
//     PlcTask Inputs/IO.ET02_Input[1] @bit 5 <-> Channel 6/Input
//     PlcTask Inputs/IO.ET02_Input[1] @bit 6 <-> Channel 7/Input
//     PlcTask Inputs/IO.ET02_Input[1] @bit 7 <-> Channel 8/Input
//     PlcTask Inputs/IO.ET02_Input[1] @bit 8 <-> Channel 9/Input
//     PlcTask Inputs/IO.ET02_Input[1] <-> Channel 1/Input
//   LS21002/LS21002 Instance <-> Device 1 (EtherCAT)/Term 16 (EK1200)/Term 29 (EK1122)/Term 41 (EK1100)/Term 43 (EL1889)
//     PlcTask Inputs/GVL_Standard.fbEhterCATSlaveMonitor[2].axIState[2] <-> WcState/WcState
//     PlcTask Inputs/IO.ET02_Input[2] @bit 9 <-> Channel 10/Input
//     PlcTask Inputs/IO.ET02_Input[2] @bit 10 <-> Channel 11/Input
//     PlcTask Inputs/IO.ET02_Input[2] @bit 11 <-> Channel 12/Input
//     PlcTask Inputs/IO.ET02_Input[2] @bit 12 <-> Channel 13/Input
//     PlcTask Inputs/IO.ET02_Input[2] @bit 13 <-> Channel 14/Input
//     PlcTask Inputs/IO.ET02_Input[2] @bit 14 <-> Channel 15/Input
//     PlcTask Inputs/IO.ET02_Input[2] @bit 15 <-> Channel 16/Input
//     PlcTask Inputs/IO.ET02_Input[2] @bit 1 <-> Channel 2/Input
//     PlcTask Inputs/IO.ET02_Input[2] @bit 2 <-> Channel 3/Input
//     PlcTask Inputs/IO.ET02_Input[2] @bit 3 <-> Channel 4/Input
//     PlcTask Inputs/IO.ET02_Input[2] @bit 4 <-> Channel 5/Input
//     PlcTask Inputs/IO.ET02_Input[2] @bit 5 <-> Channel 6/Input
//     PlcTask Inputs/IO.ET02_Input[2] @bit 6 <-> Channel 7/Input
//     PlcTask Inputs/IO.ET02_Input[2] @bit 7 <-> Channel 8/Input
//     PlcTask Inputs/IO.ET02_Input[2] @bit 8 <-> Channel 9/Input
//     PlcTask Inputs/IO.ET02_Input[2] <-> Channel 1/Input
//   LS21002/LS21002 Instance <-> Device 1 (EtherCAT)/Term 16 (EK1200)/Term 29 (EK1122)/Term 41 (EK1100)/Term 44 (EL1889)
//     PlcTask Inputs/GVL_Standard.fbEhterCATSlaveMonitor[2].axIState[3] <-> WcState/WcState
//     PlcTask Inputs/IO.ET02_Input[3] @bit 9 <-> Channel 10/Input
//     PlcTask Inputs/IO.ET02_Input[3] @bit 10 <-> Channel 11/Input
//     PlcTask Inputs/IO.ET02_Input[3] @bit 11 <-> Channel 12/Input
//     PlcTask Inputs/IO.ET02_Input[3] @bit 12 <-> Channel 13/Input
//     PlcTask Inputs/IO.ET02_Input[3] @bit 13 <-> Channel 14/Input
//     PlcTask Inputs/IO.ET02_Input[3] @bit 14 <-> Channel 15/Input
//     PlcTask Inputs/IO.ET02_Input[3] @bit 15 <-> Channel 16/Input
//     PlcTask Inputs/IO.ET02_Input[3] @bit 1 <-> Channel 2/Input
//     PlcTask Inputs/IO.ET02_Input[3] @bit 2 <-> Channel 3/Input
//     PlcTask Inputs/IO.ET02_Input[3] @bit 3 <-> Channel 4/Input
//     PlcTask Inputs/IO.ET02_Input[3] @bit 4 <-> Channel 5/Input
//     PlcTask Inputs/IO.ET02_Input[3] @bit 5 <-> Channel 6/Input
//     PlcTask Inputs/IO.ET02_Input[3] @bit 6 <-> Channel 7/Input
//     PlcTask Inputs/IO.ET02_Input[3] @bit 7 <-> Channel 8/Input
//     PlcTask Inputs/IO.ET02_Input[3] @bit 8 <-> Channel 9/Input
//     PlcTask Inputs/IO.ET02_Input[3] <-> Channel 1/Input
//   LS21002/LS21002 Instance <-> Device 1 (EtherCAT)/Term 16 (EK1200)/Term 29 (EK1122)/Term 41 (EK1100)/Term 45 (EL1889)
//     PlcTask Inputs/GVL_Standard.fbEhterCATSlaveMonitor[2].axIState[4] <-> WcState/WcState
//     PlcTask Inputs/IO.ET02_Input[4] @bit 9 <-> Channel 10/Input
//     PlcTask Inputs/IO.ET02_Input[4] @bit 10 <-> Channel 11/Input
//     PlcTask Inputs/IO.ET02_Input[4] @bit 11 <-> Channel 12/Input
//     PlcTask Inputs/IO.ET02_Input[4] @bit 12 <-> Channel 13/Input
//     PlcTask Inputs/IO.ET02_Input[4] @bit 13 <-> Channel 14/Input
//     PlcTask Inputs/IO.ET02_Input[4] @bit 14 <-> Channel 15/Input
//     PlcTask Inputs/IO.ET02_Input[4] @bit 15 <-> Channel 16/Input
//     PlcTask Inputs/IO.ET02_Input[4] @bit 1 <-> Channel 2/Input
//     PlcTask Inputs/IO.ET02_Input[4] @bit 2 <-> Channel 3/Input
//     PlcTask Inputs/IO.ET02_Input[4] @bit 3 <-> Channel 4/Input
//     PlcTask Inputs/IO.ET02_Input[4] @bit 4 <-> Channel 5/Input
//     PlcTask Inputs/IO.ET02_Input[4] @bit 5 <-> Channel 6/Input
//     PlcTask Inputs/IO.ET02_Input[4] @bit 6 <-> Channel 7/Input
//     PlcTask Inputs/IO.ET02_Input[4] @bit 7 <-> Channel 8/Input
//     PlcTask Inputs/IO.ET02_Input[4] @bit 8 <-> Channel 9/Input
//     PlcTask Inputs/IO.ET02_Input[4] <-> Channel 1/Input
//   LS21002/LS21002 Instance <-> Device 1 (EtherCAT)/Term 16 (EK1200)/Term 29 (EK1122)/Term 41 (EK1100)/Term 46 (EL1889)
//     PlcTask Inputs/GVL_Standard.fbEhterCATSlaveMonitor[2].axIState[5] <-> WcState/WcState
//     PlcTask Inputs/IO.ET02_Input[5] @bit 9 <-> Channel 10/Input
//     PlcTask Inputs/IO.ET02_Input[5] @bit 10 <-> Channel 11/Input
//     PlcTask Inputs/IO.ET02_Input[5] @bit 11 <-> Channel 12/Input
//     PlcTask Inputs/IO.ET02_Input[5] @bit 12 <-> Channel 13/Input
//     PlcTask Inputs/IO.ET02_Input[5] @bit 13 <-> Channel 14/Input
//     PlcTask Inputs/IO.ET02_Input[5] @bit 14 <-> Channel 15/Input
//     PlcTask Inputs/IO.ET02_Input[5] @bit 15 <-> Channel 16/Input
//     PlcTask Inputs/IO.ET02_Input[5] @bit 1 <-> Channel 2/Input
//     PlcTask Inputs/IO.ET02_Input[5] @bit 2 <-> Channel 3/Input
//     PlcTask Inputs/IO.ET02_Input[5] @bit 3 <-> Channel 4/Input
//     PlcTask Inputs/IO.ET02_Input[5] @bit 4 <-> Channel 5/Input
//     PlcTask Inputs/IO.ET02_Input[5] @bit 5 <-> Channel 6/Input
//     PlcTask Inputs/IO.ET02_Input[5] @bit 6 <-> Channel 7/Input
//     PlcTask Inputs/IO.ET02_Input[5] @bit 7 <-> Channel 8/Input
//     PlcTask Inputs/IO.ET02_Input[5] @bit 8 <-> Channel 9/Input
//     PlcTask Inputs/IO.ET02_Input[5] <-> Channel 1/Input
//   LS21002/LS21002 Instance <-> Device 1 (EtherCAT)/Term 16 (EK1200)/Term 29 (EK1122)/Term 41 (EK1100)/Term 47 (EL1889)
//     PlcTask Inputs/GVL_Standard.fbEhterCATSlaveMonitor[2].axIState[6] <-> WcState/WcState
//     PlcTask Inputs/IO.ET02_Input[6] @bit 9 <-> Channel 10/Input
//     PlcTask Inputs/IO.ET02_Input[6] @bit 10 <-> Channel 11/Input
//     PlcTask Inputs/IO.ET02_Input[6] @bit 11 <-> Channel 12/Input
//     PlcTask Inputs/IO.ET02_Input[6] @bit 12 <-> Channel 13/Input
//     PlcTask Inputs/IO.ET02_Input[6] @bit 13 <-> Channel 14/Input
//     PlcTask Inputs/IO.ET02_Input[6] @bit 14 <-> Channel 15/Input
//     PlcTask Inputs/IO.ET02_Input[6] @bit 15 <-> Channel 16/Input
//     PlcTask Inputs/IO.ET02_Input[6] @bit 1 <-> Channel 2/Input
//     PlcTask Inputs/IO.ET02_Input[6] @bit 2 <-> Channel 3/Input
//     PlcTask Inputs/IO.ET02_Input[6] @bit 3 <-> Channel 4/Input
//     PlcTask Inputs/IO.ET02_Input[6] @bit 4 <-> Channel 5/Input
//     PlcTask Inputs/IO.ET02_Input[6] @bit 5 <-> Channel 6/Input
//     PlcTask Inputs/IO.ET02_Input[6] @bit 6 <-> Channel 7/Input
//     PlcTask Inputs/IO.ET02_Input[6] @bit 7 <-> Channel 8/Input
//     PlcTask Inputs/IO.ET02_Input[6] @bit 8 <-> Channel 9/Input
//     PlcTask Inputs/IO.ET02_Input[6] <-> Channel 1/Input
//   LS21002/LS21002 Instance <-> Device 1 (EtherCAT)/Term 16 (EK1200)/Term 29 (EK1122)/Term 41 (EK1100)/Term 48 (EL2889)
//     PlcTask Inputs/GVL_Standard.fbEhterCATSlaveMonitor[2].axIState[7] <-> WcState/WcState
//     PlcTask Outputs/IO.ET02_Output[1] @bit 9 <-> Channel 10/Output
//     PlcTask Outputs/IO.ET02_Output[1] @bit 10 <-> Channel 11/Output
//     PlcTask Outputs/IO.ET02_Output[1] @bit 11 <-> Channel 12/Output
//     PlcTask Outputs/IO.ET02_Output[1] @bit 12 <-> Channel 13/Output
//     PlcTask Outputs/IO.ET02_Output[1] @bit 13 <-> Channel 14/Output
//     PlcTask Outputs/IO.ET02_Output[1] @bit 14 <-> Channel 15/Output
//     PlcTask Outputs/IO.ET02_Output[1] @bit 15 <-> Channel 16/Output
//     PlcTask Outputs/IO.ET02_Output[1] @bit 1 <-> Channel 2/Output
//     PlcTask Outputs/IO.ET02_Output[1] @bit 2 <-> Channel 3/Output
//     PlcTask Outputs/IO.ET02_Output[1] @bit 3 <-> Channel 4/Output
//     PlcTask Outputs/IO.ET02_Output[1] @bit 4 <-> Channel 5/Output
//     PlcTask Outputs/IO.ET02_Output[1] @bit 5 <-> Channel 6/Output
//     PlcTask Outputs/IO.ET02_Output[1] @bit 6 <-> Channel 7/Output
//     PlcTask Outputs/IO.ET02_Output[1] @bit 7 <-> Channel 8/Output
//     PlcTask Outputs/IO.ET02_Output[1] @bit 8 <-> Channel 9/Output
//     PlcTask Outputs/IO.ET02_Output[1] <-> Channel 1/Output
//   LS21002/LS21002 Instance <-> Device 1 (EtherCAT)/Term 16 (EK1200)/Term 29 (EK1122)/Term 41 (EK1100)/Term 49 (EL2889)
//     PlcTask Inputs/GVL_Standard.fbEhterCATSlaveMonitor[2].axIState[8] <-> WcState/WcState
//     PlcTask Outputs/IO.ET02_Output[2] @bit 9 <-> Channel 10/Output
//     PlcTask Outputs/IO.ET02_Output[2] @bit 10 <-> Channel 11/Output
//     PlcTask Outputs/IO.ET02_Output[2] @bit 11 <-> Channel 12/Output
//     PlcTask Outputs/IO.ET02_Output[2] @bit 12 <-> Channel 13/Output
//     PlcTask Outputs/IO.ET02_Output[2] @bit 13 <-> Channel 14/Output
//     PlcTask Outputs/IO.ET02_Output[2] @bit 14 <-> Channel 15/Output
//     PlcTask Outputs/IO.ET02_Output[2] @bit 15 <-> Channel 16/Output
//     PlcTask Outputs/IO.ET02_Output[2] @bit 1 <-> Channel 2/Output
//     PlcTask Outputs/IO.ET02_Output[2] @bit 2 <-> Channel 3/Output
//     PlcTask Outputs/IO.ET02_Output[2] @bit 3 <-> Channel 4/Output
//     PlcTask Outputs/IO.ET02_Output[2] @bit 4 <-> Channel 5/Output
//     PlcTask Outputs/IO.ET02_Output[2] @bit 5 <-> Channel 6/Output
//     PlcTask Outputs/IO.ET02_Output[2] @bit 6 <-> Channel 7/Output
//     PlcTask Outputs/IO.ET02_Output[2] @bit 7 <-> Channel 8/Output
//     PlcTask Outputs/IO.ET02_Output[2] @bit 8 <-> Channel 9/Output
//     PlcTask Outputs/IO.ET02_Output[2] <-> Channel 1/Output
//   LS21002/LS21002 Instance <-> Device 1 (EtherCAT)/Term 16 (EK1200)/Term 29 (EK1122)/Term 41 (EK1100)/Term 50 (EL2889)
//     PlcTask Inputs/GVL_Standard.fbEhterCATSlaveMonitor[2].axIState[9] <-> WcState/WcState
//     PlcTask Outputs/IO.ET02_Output[3] @bit 9 <-> Channel 10/Output
//     PlcTask Outputs/IO.ET02_Output[3] @bit 10 <-> Channel 11/Output
//     PlcTask Outputs/IO.ET02_Output[3] @bit 11 <-> Channel 12/Output
//     PlcTask Outputs/IO.ET02_Output[3] @bit 12 <-> Channel 13/Output
//     PlcTask Outputs/IO.ET02_Output[3] @bit 13 <-> Channel 14/Output
//     PlcTask Outputs/IO.ET02_Output[3] @bit 14 <-> Channel 15/Output
//     PlcTask Outputs/IO.ET02_Output[3] @bit 15 <-> Channel 16/Output
//     PlcTask Outputs/IO.ET02_Output[3] @bit 1 <-> Channel 2/Output
//     PlcTask Outputs/IO.ET02_Output[3] @bit 2 <-> Channel 3/Output
//     PlcTask Outputs/IO.ET02_Output[3] @bit 3 <-> Channel 4/Output
//     PlcTask Outputs/IO.ET02_Output[3] @bit 4 <-> Channel 5/Output
//     PlcTask Outputs/IO.ET02_Output[3] @bit 5 <-> Channel 6/Output
//     PlcTask Outputs/IO.ET02_Output[3] @bit 6 <-> Channel 7/Output
//     PlcTask Outputs/IO.ET02_Output[3] @bit 7 <-> Channel 8/Output
//     PlcTask Outputs/IO.ET02_Output[3] @bit 8 <-> Channel 9/Output
//     PlcTask Outputs/IO.ET02_Output[3] <-> Channel 1/Output
//   LS21002/LS21002 Instance <-> Device 1 (EtherCAT)/Term 16 (EK1200)/Term 29 (EK1122)/Term 41 (EK1100)/Term 51 (EL2889)
//     PlcTask Inputs/GVL_Standard.fbEhterCATSlaveMonitor[2].axIState[10] <-> WcState/WcState
//     PlcTask Outputs/IO.ET02_Output[4] @bit 9 <-> Channel 10/Output
//     PlcTask Outputs/IO.ET02_Output[4] @bit 10 <-> Channel 11/Output
//     PlcTask Outputs/IO.ET02_Output[4] @bit 11 <-> Channel 12/Output
//     PlcTask Outputs/IO.ET02_Output[4] @bit 12 <-> Channel 13/Output
//     PlcTask Outputs/IO.ET02_Output[4] @bit 13 <-> Channel 14/Output
//     PlcTask Outputs/IO.ET02_Output[4] @bit 14 <-> Channel 15/Output
//     PlcTask Outputs/IO.ET02_Output[4] @bit 15 <-> Channel 16/Output
//     PlcTask Outputs/IO.ET02_Output[4] @bit 1 <-> Channel 2/Output
//     PlcTask Outputs/IO.ET02_Output[4] @bit 2 <-> Channel 3/Output
//     PlcTask Outputs/IO.ET02_Output[4] @bit 3 <-> Channel 4/Output
//     PlcTask Outputs/IO.ET02_Output[4] @bit 4 <-> Channel 5/Output
//     PlcTask Outputs/IO.ET02_Output[4] @bit 5 <-> Channel 6/Output
//     PlcTask Outputs/IO.ET02_Output[4] @bit 6 <-> Channel 7/Output
//     PlcTask Outputs/IO.ET02_Output[4] @bit 7 <-> Channel 8/Output
//     PlcTask Outputs/IO.ET02_Output[4] @bit 8 <-> Channel 9/Output
//     PlcTask Outputs/IO.ET02_Output[4] <-> Channel 1/Output
//   LS21002/LS21002 Instance <-> Device 1 (EtherCAT)/Term 16 (EK1200)/Term 29 (EK1122)/Term 95 (EK1100)/Term 96 (EL1889)
//     PlcTask Inputs/GVL_Standard.fbEhterCATSlaveMonitor[4].axIState[1] <-> WcState/WcState
//     PlcTask Inputs/IO.ET04_Input[1] @bit 9 <-> Channel 10/Input
//     PlcTask Inputs/IO.ET04_Input[1] @bit 10 <-> Channel 11/Input
//     PlcTask Inputs/IO.ET04_Input[1] @bit 11 <-> Channel 12/Input
//     PlcTask Inputs/IO.ET04_Input[1] @bit 12 <-> Channel 13/Input
//     PlcTask Inputs/IO.ET04_Input[1] @bit 13 <-> Channel 14/Input
//     PlcTask Inputs/IO.ET04_Input[1] @bit 14 <-> Channel 15/Input
//     PlcTask Inputs/IO.ET04_Input[1] @bit 15 <-> Channel 16/Input
//     PlcTask Inputs/IO.ET04_Input[1] @bit 1 <-> Channel 2/Input
//     PlcTask Inputs/IO.ET04_Input[1] @bit 2 <-> Channel 3/Input
//     PlcTask Inputs/IO.ET04_Input[1] @bit 3 <-> Channel 4/Input
//     PlcTask Inputs/IO.ET04_Input[1] @bit 4 <-> Channel 5/Input
//     PlcTask Inputs/IO.ET04_Input[1] @bit 5 <-> Channel 6/Input
//     PlcTask Inputs/IO.ET04_Input[1] @bit 6 <-> Channel 7/Input
//     PlcTask Inputs/IO.ET04_Input[1] @bit 7 <-> Channel 8/Input
//     PlcTask Inputs/IO.ET04_Input[1] @bit 8 <-> Channel 9/Input
//     PlcTask Inputs/IO.ET04_Input[1] <-> Channel 1/Input
//   LS21002/LS21002 Instance <-> Device 1 (EtherCAT)/Term 16 (EK1200)/Term 29 (EK1122)/Term 95 (EK1100)/Term 97 (EL1889)
//     PlcTask Inputs/GVL_Standard.fbEhterCATSlaveMonitor[4].axIState[2] <-> WcState/WcState
//     PlcTask Inputs/IO.ET04_Input[2] @bit 9 <-> Channel 10/Input
//     PlcTask Inputs/IO.ET04_Input[2] @bit 10 <-> Channel 11/Input
//     PlcTask Inputs/IO.ET04_Input[2] @bit 11 <-> Channel 12/Input
//     PlcTask Inputs/IO.ET04_Input[2] @bit 12 <-> Channel 13/Input
//     PlcTask Inputs/IO.ET04_Input[2] @bit 13 <-> Channel 14/Input
//     PlcTask Inputs/IO.ET04_Input[2] @bit 14 <-> Channel 15/Input
//     PlcTask Inputs/IO.ET04_Input[2] @bit 15 <-> Channel 16/Input
//     PlcTask Inputs/IO.ET04_Input[2] @bit 1 <-> Channel 2/Input
//     PlcTask Inputs/IO.ET04_Input[2] @bit 2 <-> Channel 3/Input
//     PlcTask Inputs/IO.ET04_Input[2] @bit 3 <-> Channel 4/Input
//     PlcTask Inputs/IO.ET04_Input[2] @bit 4 <-> Channel 5/Input
//     PlcTask Inputs/IO.ET04_Input[2] @bit 5 <-> Channel 6/Input
//     PlcTask Inputs/IO.ET04_Input[2] @bit 6 <-> Channel 7/Input
//     PlcTask Inputs/IO.ET04_Input[2] @bit 7 <-> Channel 8/Input
//     PlcTask Inputs/IO.ET04_Input[2] @bit 8 <-> Channel 9/Input
//     PlcTask Inputs/IO.ET04_Input[2] <-> Channel 1/Input
//   LS21002/LS21002 Instance <-> Device 1 (EtherCAT)/Term 16 (EK1200)/Term 29 (EK1122)/Term 95 (EK1100)/Term 98 (EL2889)
//     PlcTask Inputs/GVL_Standard.fbEhterCATSlaveMonitor[4].axIState[3] <-> WcState/WcState
//     PlcTask Outputs/IO.ET04_Output[1] @bit 9 <-> Channel 10/Output
//     PlcTask Outputs/IO.ET04_Output[1] @bit 10 <-> Channel 11/Output
//     PlcTask Outputs/IO.ET04_Output[1] @bit 11 <-> Channel 12/Output
//     PlcTask Outputs/IO.ET04_Output[1] @bit 12 <-> Channel 13/Output
//     PlcTask Outputs/IO.ET04_Output[1] @bit 13 <-> Channel 14/Output
//     PlcTask Outputs/IO.ET04_Output[1] @bit 14 <-> Channel 15/Output
//     PlcTask Outputs/IO.ET04_Output[1] @bit 15 <-> Channel 16/Output
//     PlcTask Outputs/IO.ET04_Output[1] @bit 1 <-> Channel 2/Output
//     PlcTask Outputs/IO.ET04_Output[1] @bit 2 <-> Channel 3/Output
//     PlcTask Outputs/IO.ET04_Output[1] @bit 3 <-> Channel 4/Output
//     PlcTask Outputs/IO.ET04_Output[1] @bit 4 <-> Channel 5/Output
//     PlcTask Outputs/IO.ET04_Output[1] @bit 5 <-> Channel 6/Output
//     PlcTask Outputs/IO.ET04_Output[1] @bit 6 <-> Channel 7/Output
//     PlcTask Outputs/IO.ET04_Output[1] @bit 7 <-> Channel 8/Output
//     PlcTask Outputs/IO.ET04_Output[1] @bit 8 <-> Channel 9/Output
//     PlcTask Outputs/IO.ET04_Output[1] <-> Channel 1/Output
//   LS21002/LS21002 Instance <-> Device 1 (EtherCAT)/Term 16 (EK1200)/Term 29 (EK1122)/Term 95 (EK1100)/Term 99 (EL2889)
//     PlcTask Inputs/GVL_Standard.fbEhterCATSlaveMonitor[4].axIState[4] <-> WcState/WcState
//     PlcTask Outputs/IO.ET04_Output[2] @bit 9 <-> Channel 10/Output
//     PlcTask Outputs/IO.ET04_Output[2] @bit 10 <-> Channel 11/Output
//     PlcTask Outputs/IO.ET04_Output[2] @bit 11 <-> Channel 12/Output
//     PlcTask Outputs/IO.ET04_Output[2] @bit 12 <-> Channel 13/Output
//     PlcTask Outputs/IO.ET04_Output[2] @bit 13 <-> Channel 14/Output
//     PlcTask Outputs/IO.ET04_Output[2] @bit 14 <-> Channel 15/Output
//     PlcTask Outputs/IO.ET04_Output[2] @bit 15 <-> Channel 16/Output
//     PlcTask Outputs/IO.ET04_Output[2] @bit 1 <-> Channel 2/Output
//     PlcTask Outputs/IO.ET04_Output[2] @bit 2 <-> Channel 3/Output
//     PlcTask Outputs/IO.ET04_Output[2] @bit 3 <-> Channel 4/Output
//     PlcTask Outputs/IO.ET04_Output[2] @bit 4 <-> Channel 5/Output
//     PlcTask Outputs/IO.ET04_Output[2] @bit 5 <-> Channel 6/Output
//     PlcTask Outputs/IO.ET04_Output[2] @bit 6 <-> Channel 7/Output
//     PlcTask Outputs/IO.ET04_Output[2] @bit 7 <-> Channel 8/Output
//     PlcTask Outputs/IO.ET04_Output[2] @bit 8 <-> Channel 9/Output
//     PlcTask Outputs/IO.ET04_Output[2] <-> Channel 1/Output
//   LS21002/LS21002 Instance <-> Device 1 (EtherCAT)/Term 16 (EK1200)/Term 3 (EL1889)
//     PlcTask Inputs/GVL_Standard.fbEhterCATSlaveMonitor[1].axIState[2] <-> WcState/WcState
//     PlcTask Inputs/IO.ET01_Input[2] @bit 9 <-> Channel 10/Input
//     PlcTask Inputs/IO.ET01_Input[2] @bit 10 <-> Channel 11/Input
//     PlcTask Inputs/IO.ET01_Input[2] @bit 11 <-> Channel 12/Input
//     PlcTask Inputs/IO.ET01_Input[2] @bit 12 <-> Channel 13/Input
//     PlcTask Inputs/IO.ET01_Input[2] @bit 13 <-> Channel 14/Input
//     PlcTask Inputs/IO.ET01_Input[2] @bit 14 <-> Channel 15/Input
//     PlcTask Inputs/IO.ET01_Input[2] @bit 15 <-> Channel 16/Input
//     PlcTask Inputs/IO.ET01_Input[2] @bit 1 <-> Channel 2/Input
//     PlcTask Inputs/IO.ET01_Input[2] @bit 2 <-> Channel 3/Input
//     PlcTask Inputs/IO.ET01_Input[2] @bit 3 <-> Channel 4/Input
//     PlcTask Inputs/IO.ET01_Input[2] @bit 4 <-> Channel 5/Input
//     PlcTask Inputs/IO.ET01_Input[2] @bit 5 <-> Channel 6/Input
//     PlcTask Inputs/IO.ET01_Input[2] @bit 6 <-> Channel 7/Input
//     PlcTask Inputs/IO.ET01_Input[2] @bit 7 <-> Channel 8/Input
//     PlcTask Inputs/IO.ET01_Input[2] @bit 8 <-> Channel 9/Input
//     PlcTask Inputs/IO.ET01_Input[2] <-> Channel 1/Input
//   LS21002/LS21002 Instance <-> Device 1 (EtherCAT)/Term 16 (EK1200)/Term 4 (EL1889)
//     PlcTask Inputs/GVL_Standard.fbEhterCATSlaveMonitor[1].axIState[3] <-> WcState/WcState
//     PlcTask Inputs/IO.ET01_Input[3] @bit 9 <-> Channel 10/Input
//     PlcTask Inputs/IO.ET01_Input[3] @bit 10 <-> Channel 11/Input
//     PlcTask Inputs/IO.ET01_Input[3] @bit 11 <-> Channel 12/Input
//     PlcTask Inputs/IO.ET01_Input[3] @bit 12 <-> Channel 13/Input
//     PlcTask Inputs/IO.ET01_Input[3] @bit 13 <-> Channel 14/Input
//     PlcTask Inputs/IO.ET01_Input[3] @bit 14 <-> Channel 15/Input
//     PlcTask Inputs/IO.ET01_Input[3] @bit 15 <-> Channel 16/Input
//     PlcTask Inputs/IO.ET01_Input[3] @bit 1 <-> Channel 2/Input
//     PlcTask Inputs/IO.ET01_Input[3] @bit 2 <-> Channel 3/Input
//     PlcTask Inputs/IO.ET01_Input[3] @bit 3 <-> Channel 4/Input
//     PlcTask Inputs/IO.ET01_Input[3] @bit 4 <-> Channel 5/Input
//     PlcTask Inputs/IO.ET01_Input[3] @bit 5 <-> Channel 6/Input
//     PlcTask Inputs/IO.ET01_Input[3] @bit 6 <-> Channel 7/Input
//     PlcTask Inputs/IO.ET01_Input[3] @bit 7 <-> Channel 8/Input
//     PlcTask Inputs/IO.ET01_Input[3] @bit 8 <-> Channel 9/Input
//     PlcTask Inputs/IO.ET01_Input[3] <-> Channel 1/Input
//   LS21002/LS21002 Instance <-> Device 1 (EtherCAT)/Term 16 (EK1200)/Term 5 (EL1889)
//     PlcTask Inputs/GVL_Standard.fbEhterCATSlaveMonitor[1].axIState[4] <-> WcState/WcState
//     PlcTask Inputs/IO.ET01_Input[4] @bit 9 <-> Channel 10/Input
//     PlcTask Inputs/IO.ET01_Input[4] @bit 10 <-> Channel 11/Input
//     PlcTask Inputs/IO.ET01_Input[4] @bit 11 <-> Channel 12/Input
//     PlcTask Inputs/IO.ET01_Input[4] @bit 12 <-> Channel 13/Input
//     PlcTask Inputs/IO.ET01_Input[4] @bit 13 <-> Channel 14/Input
//     PlcTask Inputs/IO.ET01_Input[4] @bit 14 <-> Channel 15/Input
//     PlcTask Inputs/IO.ET01_Input[4] @bit 15 <-> Channel 16/Input
//     PlcTask Inputs/IO.ET01_Input[4] @bit 1 <-> Channel 2/Input
//     PlcTask Inputs/IO.ET01_Input[4] @bit 2 <-> Channel 3/Input
//     PlcTask Inputs/IO.ET01_Input[4] @bit 3 <-> Channel 4/Input
//     PlcTask Inputs/IO.ET01_Input[4] @bit 4 <-> Channel 5/Input
//     PlcTask Inputs/IO.ET01_Input[4] @bit 5 <-> Channel 6/Input
//     PlcTask Inputs/IO.ET01_Input[4] @bit 6 <-> Channel 7/Input
//     PlcTask Inputs/IO.ET01_Input[4] @bit 7 <-> Channel 8/Input
//     PlcTask Inputs/IO.ET01_Input[4] @bit 8 <-> Channel 9/Input
//     PlcTask Inputs/IO.ET01_Input[4] <-> Channel 1/Input
//   LS21002/LS21002 Instance <-> Device 1 (EtherCAT)/Term 16 (EK1200)/Term 6 (EL1889)
//     PlcTask Inputs/GVL_Standard.fbEhterCATSlaveMonitor[1].axIState[5] <-> WcState/WcState
//     PlcTask Inputs/IO.ET01_Input[5] @bit 9 <-> Channel 10/Input
//     PlcTask Inputs/IO.ET01_Input[5] @bit 10 <-> Channel 11/Input
//     PlcTask Inputs/IO.ET01_Input[5] @bit 11 <-> Channel 12/Input
//     PlcTask Inputs/IO.ET01_Input[5] @bit 12 <-> Channel 13/Input
//     PlcTask Inputs/IO.ET01_Input[5] @bit 13 <-> Channel 14/Input
//     PlcTask Inputs/IO.ET01_Input[5] @bit 14 <-> Channel 15/Input
//     PlcTask Inputs/IO.ET01_Input[5] @bit 15 <-> Channel 16/Input
//     PlcTask Inputs/IO.ET01_Input[5] @bit 1 <-> Channel 2/Input
//     PlcTask Inputs/IO.ET01_Input[5] @bit 2 <-> Channel 3/Input
//     PlcTask Inputs/IO.ET01_Input[5] @bit 3 <-> Channel 4/Input
//     PlcTask Inputs/IO.ET01_Input[5] @bit 4 <-> Channel 5/Input
//     PlcTask Inputs/IO.ET01_Input[5] @bit 5 <-> Channel 6/Input
//     PlcTask Inputs/IO.ET01_Input[5] @bit 6 <-> Channel 7/Input
//     PlcTask Inputs/IO.ET01_Input[5] @bit 7 <-> Channel 8/Input
//     PlcTask Inputs/IO.ET01_Input[5] @bit 8 <-> Channel 9/Input
//     PlcTask Inputs/IO.ET01_Input[5] <-> Channel 1/Input
//   LS21002/LS21002 Instance <-> Device 1 (EtherCAT)/Term 16 (EK1200)/Term 7 (EL1889)
//     PlcTask Inputs/GVL_Standard.fbEhterCATSlaveMonitor[1].axIState[6] <-> WcState/WcState
//     PlcTask Inputs/IO.ET01_Input[6] @bit 9 <-> Channel 10/Input
//     PlcTask Inputs/IO.ET01_Input[6] @bit 10 <-> Channel 11/Input
//     PlcTask Inputs/IO.ET01_Input[6] @bit 11 <-> Channel 12/Input
//     PlcTask Inputs/IO.ET01_Input[6] @bit 12 <-> Channel 13/Input
//     PlcTask Inputs/IO.ET01_Input[6] @bit 13 <-> Channel 14/Input
//     PlcTask Inputs/IO.ET01_Input[6] @bit 14 <-> Channel 15/Input
//     PlcTask Inputs/IO.ET01_Input[6] @bit 15 <-> Channel 16/Input
//     PlcTask Inputs/IO.ET01_Input[6] @bit 1 <-> Channel 2/Input
//     PlcTask Inputs/IO.ET01_Input[6] @bit 2 <-> Channel 3/Input
//     PlcTask Inputs/IO.ET01_Input[6] @bit 3 <-> Channel 4/Input
//     PlcTask Inputs/IO.ET01_Input[6] @bit 4 <-> Channel 5/Input
//     PlcTask Inputs/IO.ET01_Input[6] @bit 5 <-> Channel 6/Input
//     PlcTask Inputs/IO.ET01_Input[6] @bit 6 <-> Channel 7/Input
//     PlcTask Inputs/IO.ET01_Input[6] @bit 7 <-> Channel 8/Input
//     PlcTask Inputs/IO.ET01_Input[6] @bit 8 <-> Channel 9/Input
//     PlcTask Inputs/IO.ET01_Input[6] <-> Channel 1/Input
//   LS21002/LS21002 Instance <-> Device 1 (EtherCAT)/Term 16 (EK1200)/Term 8 (EL2889)
//     PlcTask Inputs/GVL_Standard.fbEhterCATSlaveMonitor[1].axIState[7] <-> WcState/WcState
//     PlcTask Outputs/IO.ET01_Output[1] @bit 9 <-> Channel 10/Output
//     PlcTask Outputs/IO.ET01_Output[1] @bit 10 <-> Channel 11/Output
//     PlcTask Outputs/IO.ET01_Output[1] @bit 11 <-> Channel 12/Output
//     PlcTask Outputs/IO.ET01_Output[1] @bit 12 <-> Channel 13/Output
//     PlcTask Outputs/IO.ET01_Output[1] @bit 13 <-> Channel 14/Output
//     PlcTask Outputs/IO.ET01_Output[1] @bit 14 <-> Channel 15/Output
//     PlcTask Outputs/IO.ET01_Output[1] @bit 15 <-> Channel 16/Output
//     PlcTask Outputs/IO.ET01_Output[1] @bit 1 <-> Channel 2/Output
//     PlcTask Outputs/IO.ET01_Output[1] @bit 2 <-> Channel 3/Output
//     PlcTask Outputs/IO.ET01_Output[1] @bit 3 <-> Channel 4/Output
//     PlcTask Outputs/IO.ET01_Output[1] @bit 4 <-> Channel 5/Output
//     PlcTask Outputs/IO.ET01_Output[1] @bit 5 <-> Channel 6/Output
//     PlcTask Outputs/IO.ET01_Output[1] @bit 6 <-> Channel 7/Output
//     PlcTask Outputs/IO.ET01_Output[1] @bit 7 <-> Channel 8/Output
//     PlcTask Outputs/IO.ET01_Output[1] @bit 8 <-> Channel 9/Output
//     PlcTask Outputs/IO.ET01_Output[1] <-> Channel 1/Output
//   LS21002/LS21002 Instance <-> Device 1 (EtherCAT)/Term 16 (EK1200)/Term 9 (EL2889)
//     PlcTask Inputs/GVL_Standard.fbEhterCATSlaveMonitor[1].axIState[8] <-> WcState/WcState
//     PlcTask Outputs/IO.ET01_Output[2] @bit 9 <-> Channel 10/Output
//     PlcTask Outputs/IO.ET01_Output[2] @bit 10 <-> Channel 11/Output
//     PlcTask Outputs/IO.ET01_Output[2] @bit 11 <-> Channel 12/Output
//     PlcTask Outputs/IO.ET01_Output[2] @bit 12 <-> Channel 13/Output
//     PlcTask Outputs/IO.ET01_Output[2] @bit 13 <-> Channel 14/Output
//     PlcTask Outputs/IO.ET01_Output[2] @bit 14 <-> Channel 15/Output
//     PlcTask Outputs/IO.ET01_Output[2] @bit 15 <-> Channel 16/Output
//     PlcTask Outputs/IO.ET01_Output[2] @bit 1 <-> Channel 2/Output
//     PlcTask Outputs/IO.ET01_Output[2] @bit 2 <-> Channel 3/Output
//     PlcTask Outputs/IO.ET01_Output[2] @bit 3 <-> Channel 4/Output
//     PlcTask Outputs/IO.ET01_Output[2] @bit 4 <-> Channel 5/Output
//     PlcTask Outputs/IO.ET01_Output[2] @bit 5 <-> Channel 6/Output
//     PlcTask Outputs/IO.ET01_Output[2] @bit 6 <-> Channel 7/Output
//     PlcTask Outputs/IO.ET01_Output[2] @bit 7 <-> Channel 8/Output
//     PlcTask Outputs/IO.ET01_Output[2] @bit 8 <-> Channel 9/Output
//     PlcTask Outputs/IO.ET01_Output[2] <-> Channel 1/Output
//   LS21002/LS21002 Instance <-> NC-Task 1 SAF/Axes/Axis 1
//     PlcTask Inputs/CallStandard.nctrl1[1] <-> Drive/Outputs/Out/nCtrl1
//     PlcTask Inputs/CallStandard.nctrl2[1] <-> Drive/Outputs/Out/nCtrl2
//     PlcTask Inputs/GVL_Standard.Axis[1].NcToPlc <-> Outputs/ToPlc
//     PlcTask Outputs/GVL_Standard.Axis[1].PlcToNc <-> Inputs/FromPlc
//   LS21002/LS21002 Instance <-> NC-Task 1 SAF/Axes/Axis 10
//     PlcTask Inputs/CallStandard.nctrl1[10] <-> Drive/Outputs/Out/nCtrl1
//     PlcTask Inputs/CallStandard.nctrl2[10] <-> Drive/Outputs/Out/nCtrl2
//     PlcTask Inputs/GVL_Standard.Axis[10].NcToPlc <-> Outputs/ToPlc
//     PlcTask Outputs/GVL_Standard.Axis[10].PlcToNc <-> Inputs/FromPlc
//   LS21002/LS21002 Instance <-> NC-Task 1 SAF/Axes/Axis 11
//     PlcTask Inputs/CallStandard.nctrl1[11] <-> Drive/Outputs/Out/nCtrl1
//     PlcTask Inputs/CallStandard.nctrl2[11] <-> Drive/Outputs/Out/nCtrl2
//     PlcTask Inputs/GVL_Standard.Axis[11].NcToPlc <-> Outputs/ToPlc
//     PlcTask Outputs/GVL_Standard.Axis[11].PlcToNc <-> Inputs/FromPlc
//   LS21002/LS21002 Instance <-> NC-Task 1 SAF/Axes/Axis 12
//     PlcTask Inputs/CallStandard.nctrl1[12] <-> Drive/Outputs/Out/nCtrl1
//     PlcTask Inputs/CallStandard.nctrl2[12] <-> Drive/Outputs/Out/nCtrl2
//     PlcTask Inputs/GVL_Standard.Axis[12].NcToPlc <-> Outputs/ToPlc
//     PlcTask Outputs/GVL_Standard.Axis[12].PlcToNc <-> Inputs/FromPlc
//   LS21002/LS21002 Instance <-> NC-Task 1 SAF/Axes/Axis 13
//     PlcTask Inputs/CallStandard.nctrl1[13] <-> Drive/Outputs/Out/nCtrl1
//     PlcTask Inputs/CallStandard.nctrl2[13] <-> Drive/Outputs/Out/nCtrl2
//     PlcTask Inputs/GVL_Standard.Axis[13].NcToPlc <-> Outputs/ToPlc
//     PlcTask Outputs/GVL_Standard.Axis[13].PlcToNc <-> Inputs/FromPlc
//   LS21002/LS21002 Instance <-> NC-Task 1 SAF/Axes/Axis 14
//     PlcTask Inputs/CallStandard.nctrl1[14] <-> Drive/Outputs/Out/nCtrl1
//     PlcTask Inputs/CallStandard.nctrl2[14] <-> Drive/Outputs/Out/nCtrl2
//     PlcTask Inputs/GVL_Standard.Axis[14].NcToPlc <-> Outputs/ToPlc
//     PlcTask Outputs/GVL_Standard.Axis[14].PlcToNc <-> Inputs/FromPlc
//   LS21002/LS21002 Instance <-> NC-Task 1 SAF/Axes/Axis 15
//     PlcTask Inputs/CallStandard.nctrl1[15] <-> Drive/Outputs/Out/nCtrl1
//     PlcTask Inputs/CallStandard.nctrl2[15] <-> Drive/Outputs/Out/nCtrl2
//     PlcTask Inputs/GVL_Standard.Axis[15].NcToPlc <-> Outputs/ToPlc
//     PlcTask Outputs/GVL_Standard.Axis[15].PlcToNc <-> Inputs/FromPlc
//   LS21002/LS21002 Instance <-> NC-Task 1 SAF/Axes/Axis 16
//     PlcTask Inputs/CallStandard.nctrl1[16] <-> Drive/Outputs/Out/nCtrl1
//     PlcTask Inputs/CallStandard.nctrl2[16] <-> Drive/Outputs/Out/nCtrl2
//     PlcTask Inputs/GVL_Standard.Axis[16].NcToPlc <-> Outputs/ToPlc
//     PlcTask Outputs/GVL_Standard.Axis[16].PlcToNc <-> Inputs/FromPlc
//   LS21002/LS21002 Instance <-> NC-Task 1 SAF/Axes/Axis 17
//     PlcTask Inputs/CallStandard.nctrl1[17] <-> Drive/Outputs/Out/nCtrl1
//     PlcTask Inputs/CallStandard.nctrl2[17] <-> Drive/Outputs/Out/nCtrl2
//     PlcTask Inputs/GVL_Standard.Axis[17].NcToPlc <-> Outputs/ToPlc
//     PlcTask Outputs/GVL_Standard.Axis[17].PlcToNc <-> Inputs/FromPlc
//   LS21002/LS21002 Instance <-> NC-Task 1 SAF/Axes/Axis 18
//     PlcTask Inputs/CallStandard.nctrl1[18] <-> Drive/Outputs/Out/nCtrl1
//     PlcTask Inputs/CallStandard.nctrl2[18] <-> Drive/Outputs/Out/nCtrl2
//     PlcTask Inputs/GVL_Standard.Axis[18].NcToPlc <-> Outputs/ToPlc
//     PlcTask Outputs/GVL_Standard.Axis[18].PlcToNc <-> Inputs/FromPlc
//   LS21002/LS21002 Instance <-> NC-Task 1 SAF/Axes/Axis 19
//     PlcTask Inputs/CallStandard.nctrl1[19] <-> Drive/Outputs/Out/nCtrl1
//     PlcTask Inputs/CallStandard.nctrl2[19] <-> Drive/Outputs/Out/nCtrl2
//     PlcTask Inputs/GVL_Standard.Axis[19].NcToPlc <-> Outputs/ToPlc
//     PlcTask Outputs/GVL_Standard.Axis[19].PlcToNc <-> Inputs/FromPlc
//   LS21002/LS21002 Instance <-> NC-Task 1 SAF/Axes/Axis 2
//     PlcTask Inputs/CallStandard.nctrl1[2] <-> Drive/Outputs/Out/nCtrl1
//     PlcTask Inputs/CallStandard.nctrl2[2] <-> Drive/Outputs/Out/nCtrl2
//     PlcTask Inputs/GVL_Standard.Axis[2].NcToPlc <-> Outputs/ToPlc
//     PlcTask Outputs/GVL_Standard.Axis[2].PlcToNc <-> Inputs/FromPlc
//   LS21002/LS21002 Instance <-> NC-Task 1 SAF/Axes/Axis 3
//     PlcTask Inputs/CallStandard.nctrl1[3] <-> Drive/Outputs/Out/nCtrl1
//     PlcTask Inputs/CallStandard.nctrl2[3] <-> Drive/Outputs/Out/nCtrl2
//     PlcTask Inputs/GVL_Standard.Axis[3].NcToPlc <-> Outputs/ToPlc
//     PlcTask Outputs/GVL_Standard.Axis[3].PlcToNc <-> Inputs/FromPlc
//   LS21002/LS21002 Instance <-> NC-Task 1 SAF/Axes/Axis 4
//     PlcTask Inputs/CallStandard.nctrl1[4] <-> Drive/Outputs/Out/nCtrl1
//     PlcTask Inputs/CallStandard.nctrl2[4] <-> Drive/Outputs/Out/nCtrl2
//     PlcTask Inputs/GVL_Standard.Axis[4].NcToPlc <-> Outputs/ToPlc
//     PlcTask Outputs/GVL_Standard.Axis[4].PlcToNc <-> Inputs/FromPlc
//   LS21002/LS21002 Instance <-> NC-Task 1 SAF/Axes/Axis 5
//     PlcTask Inputs/CallStandard.nctrl1[5] <-> Drive/Outputs/Out/nCtrl1
//     PlcTask Inputs/CallStandard.nctrl2[5] <-> Drive/Outputs/Out/nCtrl2
//     PlcTask Inputs/GVL_Standard.Axis[5].NcToPlc <-> Outputs/ToPlc
//     PlcTask Outputs/GVL_Standard.Axis[5].PlcToNc <-> Inputs/FromPlc
//   LS21002/LS21002 Instance <-> NC-Task 1 SAF/Axes/Axis 6
//     PlcTask Inputs/CallStandard.nctrl1[6] <-> Drive/Outputs/Out/nCtrl1
//     PlcTask Inputs/CallStandard.nctrl2[6] <-> Drive/Outputs/Out/nCtrl2
//     PlcTask Inputs/GVL_Standard.Axis[6].NcToPlc <-> Outputs/ToPlc
//     PlcTask Outputs/GVL_Standard.Axis[6].PlcToNc <-> Inputs/FromPlc
//   LS21002/LS21002 Instance <-> NC-Task 1 SAF/Axes/Axis 7
//     PlcTask Inputs/CallStandard.nctrl1[7] <-> Drive/Outputs/Out/nCtrl1
//     PlcTask Inputs/CallStandard.nctrl2[7] <-> Drive/Outputs/Out/nCtrl2
//     PlcTask Inputs/GVL_Standard.Axis[7].NcToPlc <-> Outputs/ToPlc
//     PlcTask Outputs/GVL_Standard.Axis[7].PlcToNc <-> Inputs/FromPlc
//   LS21002/LS21002 Instance <-> NC-Task 1 SAF/Axes/Axis 8
//     PlcTask Inputs/CallStandard.nctrl1[8] <-> Drive/Outputs/Out/nCtrl1
//     PlcTask Inputs/CallStandard.nctrl2[8] <-> Drive/Outputs/Out/nCtrl2
//     PlcTask Inputs/GVL_Standard.Axis[8].NcToPlc <-> Outputs/ToPlc
//     PlcTask Outputs/GVL_Standard.Axis[8].PlcToNc <-> Inputs/FromPlc
//   LS21002/LS21002 Instance <-> NC-Task 1 SAF/Axes/Axis 9
//     PlcTask Inputs/CallStandard.nctrl1[9] <-> Drive/Outputs/Out/nCtrl1
//     PlcTask Inputs/CallStandard.nctrl2[9] <-> Drive/Outputs/Out/nCtrl2
//     PlcTask Inputs/GVL_Standard.Axis[9].NcToPlc <-> Outputs/ToPlc
//     PlcTask Outputs/GVL_Standard.Axis[9].PlcToNc <-> Inputs/FromPlc

CONFIGURATION LS21002
    RESOURCE PLC ON TwinCAT3
        TASK PlcTask(INTERVAL := T#10ms, PRIORITY := 20);
        PROGRAM MAIN WITH PlcTask : MAIN;
    END_RESOURCE
END_CONFIGURATION

// ---- DUTs/Camera/DUT_CameraSend.TcDUT
TYPE DUT_CameraSend :
STRUCT
//Camera----PLC  //[1]---工控机1  [2]---工控机2  [3]---工控机3
   iCameraAlive 	:ARRAY[1..3] OF INT; ;//0=false  1=true，  								  
   iStatus			:ARRAY[1..3] OF INT;//相机准备状态 1=就绪  2=未就绪   							 
   iCompleted		:ARRAY[1..18] OF INT;//相机拍照完成    1=完成   1<>未完成   触发前PLC清除
   iS01Result		:ARRAY[1..4]  OF  INT;//相机拍照结果， 1=OK  2=角度反  3=料反，触发前PLC清除	
   iS03Result		:ARRAY[1..16]  OF  INT;//相机拍照结果， 1=OK  2=NG，触发前PLC清除
   iS13Result		:ARRAY[1..1]  OF  INT;//相机拍照结果， 1=OK 2=NG，触发前PLC清除																	
END_STRUCT
END_TYPE

// ---- DUTs/Camera/DUT_CameraReceive.TcDUT
TYPE DUT_CameraReceive :
STRUCT
   iBoxType 	: INT; ;//1=锥底光滑身 2=圆底断崖身，  								 													
END_STRUCT
END_TYPE

// ---- DUTs/Camera/ST_CameraPara.TcDUT
TYPE ST_CameraPara :
STRUCT
	tDelay:TIME;
END_STRUCT
END_TYPE

// ---- DUTs/DUT_NCIO.TcDUT
TYPE DUT_NCIO :
STRUCT
	nDataIn1:DINT;
 (*	nDataIn2:INT;*)
	nState1:UINT;
	nState2:UINT;
	nState3:UINT;
	nState4:UINT;
	nDataIn3:INT;
	nDataIn4:INT;
	nDataIn5:INT;
	nDataIn6:INT;
	nState5:SINT;
	nState6:SINT;
	nState7:SINT;
	nState8:SINT;
	nDcInputTime:INT;
	nData   :ARRAY[1..80] OF BYTE;
	
	
END_STRUCT
END_TYPE

// ---- DUTs/DUT_NCIO_1.TcDUT
TYPE DUT_NCIO_1 :
STRUCT
	nDataIn1:DINT;
 (*	nDataIn2:INT;
	nState1:UINT;
	nState2:UINT;
	nState3:UINT;
	nState4:UINT;
	nDataIn3:INT;
	nDataIn4:INT;
	nDataIn5:INT;
	nDataIn6:INT;
	nState5:SINT;
	nState6:SINT;
	nState7:SINT;
	nState8:SINT;
	nDcInputTime:INT;*)
	nData1   :ARRAY[1..32] OF BYTE;
	
	nDataIn2:DINT;
	nData2   :ARRAY[1..72] OF BYTE;
	
	
END_STRUCT
END_TYPE

